// TIA Portal V20 export
// export: Created 2025-12-01T14:57:14.0359159Z, ExportSetting None, DisplayName Totally Integrated Automation Portal, DisplayVersion V20 Update 3, DisplayName TIA Portal Openness, DisplayVersion V20 Update 3, DisplayName TIA Portal Version Control Interface, DisplayVersion V20 Update 3, DisplayName STEP 7 Professional, DisplayVersion V20 Update 3, DisplayName STEP 7 Safety, DisplayVersion V20 Update 2, DisplayName WinCC Basic/Comfort/Advanced, DisplayVersion V20 Update 3, DisplayName WinCC Professional, DisplayVersion V20 Update 3, DisplayName WinCC Unified, DisplayVersion V20 Update 3
FUNCTION "FC810_EventosRecibidos" : Void   // FC810, LAD
TITLE = "Eventos Recibidos" - Tratamiento de los Eventos
{ S7_Optimized_Access := 'FALSE' }
AUTHOR : TRACKING
NAME : 20170707
VERSION : 4.5
// stored: AutoNumber false, SetENOAutomatically false
   VAR_INPUT
      NumJDT : UInt;
   END_VAR
   VAR_TEMP
      AtributosDeUTs : Struct   // Atributos Recibidos de las UTs
         Ruta : Array[0..20] of UInt;   // Ruta Recibida
         Etiqueta : Array[0..42] of Char;   // Etiqueta
         QUBIQA_PID : Array[0..20] of Char;   // QUBIQA - PID del Bulto
         CambiarUTDeMesa : Struct
            Origen : UInt;
            Destino : UInt;
            NOK : Bool;
            OK : Bool;
            Inicio : Bool;
            Final : Bool;
         END_STRUCT;
         AtributosTipoDeCarga : Struct
            Vacia : Bool;
            Pila : Bool;
            Remontada : Bool;
         END_STRUCT;
         Mckey : UDInt;   // Mckey
         MesaActual : UInt;   // Mesa Actual
         MesaDestino : UInt;   // Mesa Destino
         MesaIntermedia : UInt;   // Mesa Intermedia
         OrdenSalida : UInt;   // Orden de Salida
         TipoCarga : USInt;   // **** Tipo de la Carga
         Grupo : UInt;   // Grupo
         CantidadGrupo : USInt;   // Cantidad del Grupo
         PosicionGrupo : USInt;   // Posicion del Grupo
         CodigoFlejado : USInt;   // Codigo de Flejado
         CodigoEnfardado : USInt;   // Codigo de Enfradado
         CodigoEtiquetado : USInt;   // Codigo de Etiquetado
         GaliboAltura : USInt;   // Galibo - Codigo de Altura
         GaliboAnchura : USInt;   // Galibo - Codigo de Anchura
         GaliboProfundidad : USInt;   // Galibo - Codigo de Profundidad
         GaliboTaco : USInt;   // Galibo - Codigo de Taco
         GaliboHueco : USInt;   // Galibo - Codigo de Hueco
         GaliboHuecoRemontada : USInt;   // Galibo - Codigo de Hueco de Carga Remontada
         GaliboColor : USInt;   // Galibo - Codigo de Color de la Carga
         GaliboPatin : USInt;   // Galibo - Codigo de Patin
         GaliboSGA : USInt;   // Galibo - Codigo de SGA
         Presion : UInt;   // Presion de DesPaletizado o Paletizaado de Cajas de Plastico
         CotaAmarre : UInt;   // Cota de Amarre de Cajas de Plastico
         CotaAltura : UInt;   // Cota de la Altura
         CotaAnchura : UInt;   // Cota de la Anchura
         CotaProfundidad : UInt;   // Cota de la Profundidad
         Peso : UDInt;   // Peso
         PosicionDeLaEtiqueta : UInt;   // Posicion Actual de la Etiqueta
         QUBIQA_NumeroBulto : UInt;   // QUBIQA - Numero de Bulto
         QUBIQA_TotalBultos : UInt;   // QUBIQA - Numero Total de Bultos
      END_STRUCT;
      AtributosDeDispositivos : Struct   // Atributos Recibidos del Dispositivo
         TextoRecibido : Array[0..50] of Char;
         MotivoDelError : Array[0..50] of Char;   // TEXTO - Motivo del Error
         BalizaColor : "UDT_DatosBaliza";
         Tipo : UInt;   // Tipo
         Numero : UInt;   // Numero
         NuevoEstado : UInt;   // NuevoEstado
         Habilitado : UInt;
         Prioridad : UInt;
         Operacion : UInt;
         MesaHorquilla : UInt;
         MesaCargaDesCarga : UInt;
      END_STRUCT;
      VarTempUTs : Struct
         Mckey : UDInt;
         MesaActual : UInt;
         NumeroUT : UInt;
         SalidaEventoRETI : UInt;
      END_STRUCT;
      VarTempDispositivos : Struct
         Baliza : "UDT_DatosBaliza";
         Numero : UInt;
      END_STRUCT;
      DBEventosRec : Word;   // DB de Eventos Recibidos
      P_Eventos : DWord;   // Puntero al DB de Eventos Recibidos
      Evento : DWord;   // Etiqueta - Evento
      Atributo : DWord;   // Etiqueta - Atributo
      EtiquetaAtributo : DWord;   // Etiqueta - Conversion de Atributo
      NumeroEvento : UInt;   // Numero de Evento
      NumeroAtributo : UInt;   // Numero de Atributo
      Leido : UInt;
      ValorDeAtributo : UDInt;   // Valor del Atributo
      ValorDeEtiqueta : UInt;   // Valor de la Etiqueta - Conversion de Atributo
      Indice : UInt;   // Indice en el recorrido de los ARRAYs
      IndiceCBOX : UInt;
      IndiceVTDC : UInt;
      IndiceMesa : UInt;
      IndiceMaquina : UInt;
      IndiceDispositivosVarios : UInt;
      OffsetInicial : UInt;
      LonguitudTextoRecibido : UInt;
      ReturnValor : Int;
      Cero : Byte;
      JDT02_Activo : Bool;
      MesaDeJDT02 : Bool;
      DispositivoDeJDT02 : Bool;
   END_VAR
BEGIN

NETWORK
TITLE = Inicializar
/////////////////////////////////////////////////////////////////////////
/// --- Comprobar que JDT

      SET;
      R     #JDT02_Activo;
      L     "JDT1_NDB_EventosRec";  // Cogemos el DB de Eventos Recibidos
      T     #DBEventosRec;

/////////////////////////////////////////////////////////////////////////

      L     #NumJDT;
      L     2;
      <>I;
      JC    NoJdT02;

/////////////////////////////////////////////////////////////////////////

      SET;
      S     #JDT02_Activo;
      L     "JDT2_NDB_EventosRec";  // Cogemos el DB de Eventos Recibidos
      T     #DBEventosRec;

NoJdT02:NOP   0;

/////////////////////////////////////////////////////////////////////////



NETWORK
TITLE = Analizar la lista de Eventos
/////////////////////////////////////////////////////////////////////////
// Inicializar el Puntero de la Lista de Eventos

      L     0;  // Inicializar el Puntero de Eventos
      LAR2;

      OPN   DB [#DBEventosRec];  // Mirar si tiene algo el DB de Eventos Recibidos
      L     DBB [AR2, P#0.0];
      L     0;
      ==I;
      JC    NoLimpiarNada;


/////////////////////////////////////////////////////////////////////////
InicioBucle_EventosRecibidos:NOP   0;
      OPN   DB [#DBEventosRec];  // Leer el digito de Eventos Recibidos
      L     DBB [AR2, P#0.0];
      T     #Leido;

// Buscando Principio de Evento

      L     #Leido;
      L     '{';  // Inicio de Evento - '{'
      ==I;
      JC    EventosRecibidos;  // Tratar el Nuevo Evento

// Buscando el Final de la Lista de Eventos

      L     #Leido;
      L     3;  // Final de la Lista de Eventos - 0x03
      ==I;
      JC    FinalizarFuncion;  // Finalizar, ya no hay más Eventos
      L     #Leido;
      L     0;  // Final de la Lista de Eventos - 0x00 - No hay Mas
      ==I;
      JC    FinalizarFuncion;  // Finalizar, ya no hay más Eventos


/////////////////////////////////////////////////////////////////////////
FinBucle_EventosRecibidos:NOP   0;
      +AR2  P#1.0;  // Seguir recorriendo la Lista de Eventos
      JU    InicioBucle_EventosRecibidos;



NETWORK
TITLE = Distribucion de los Eventos (LIsta del DB de Conversion)
EventosRecibidos:NOP   0;

/////////////////////////////////////////////////////////////////////////
/////////////////////////////////////////////////////////////////////////
/////////////////////////////////////////////////////////////////////////
// Hay que recoger el Evento, para despues repartir
// Despues '{' va el tipo de eventos (2 Bytes)

      +AR2  P#1.0;
      OPN   DB [#DBEventosRec];
      L     DBD [AR2, P#0.0];  // Recogo el tipo de Evento (4 Caracteres)
      T     #Evento;


/////////////////////////////////////////////////////////////////////////
/////////////////////////////////////////////////////////////////////////
/////////////////////////////////////////////////////////////////////////
// Buscar numero de evento
      L     1;
      T     #NumeroEvento;
BucleDeBusqueda_NumeroDeEvento:NOP   0;

// -- Se ha encontrado el Evento Recibido
      L     "DB870_ConversorEventos".EventosRecibidos[#NumeroEvento];
      L     #Evento;
      ==D;
      JC    Encontrado_NumeroDeEvento;

// -- Final de la lista de Eventos Recibidos - No Encontrado
      L     "DB870_ConversorEventos".EventosRecibidos[#NumeroEvento];
      L     0;
      ==D;
      JC    InicioBucle_EventosRecibidos;

// --- Maximo del Array de la Lista de Eventos Recibidos - No Encontrado
      L     #NumeroEvento;
      L     "CTE_MaxArrayConversion";
      >=I;
      JC    InicioBucle_EventosRecibidos;

// --- Continuar la Busqueda
      L     #NumeroEvento;
      L     1;
      +I;
      T     #NumeroEvento;
      JU    BucleDeBusqueda_NumeroDeEvento;



NETWORK
TITLE = ----
/////////////////////////////////////////////////////////////////////////
/////////////////////////////////////////////////////////////////////////
/////////////////////////////////////////////////////////////////////////
// Distribuir dependiendo del Resultado de la Busqueda del Evento Recibido
// Para recoger los Atributos
Encontrado_NumeroDeEvento:NOP   0;
      L     #NumeroEvento;
      JL    NoExiste_NumeroDeEvento;

      JU    NoExiste_NumeroDeEvento;
      JU    Atributos_EventosDeLasUTs;  // Evento (01) - CREA
      JU    Atributos_EventosDeLasUTs;  // Evento (02) - RUTA
      JU    Atributos_EventosDeLasUTs;  // Evento (03) - DRUT
      JU    Atributos_EventosDeLasUTs;  // Evento (04) - RETI
      JU    Atributos_EventosDeLasUTs;  // Evento (05) - BORR
      JU    Atributos_EventosDeLasUTs;  // Evento (06) - DATA
      JU    Atributos_EventosDeLasUTs;  // Evento (07) - ?UT?
      JU    Atributos_EventosDeLasUTs;  // Evento (08) - MOVE
      JU    Atributos_EventosDeLasUTs;  // Evento (09) - DEMB

      JU    Atributos_EventosDeLosDispositivos;  // Evento (10) - CSTA
      JU    Atributos_EventosDeLosDispositivos;  // Evento (11) - DIDO

      JU    EventosRecibidos_Router;  // Evento (12) - ORDE
      JU    EventosRecibidos_Router;  // Evento (13) - BOET
      JU    EventosRecibidos_Router;  // Evento (14) - BOBD
      JU    EventosRecibidos_Router;  // Evento (15) - RUET
      JU    EventosRecibidos_Router;  // Evento (16) - RUES
      JU    EventosRecibidos_Router;  // Evento (17) - INIR

      JU    Atributos_EventosDeLosDispositivos;  // Evento (18) - ?ST?

      JU    EventosRecibidos_Quimarox;  // Evento (19) - QCRE
      JU    EventosRecibidos_Quimarox;  // Evento (20) - QPR?

      JU    EventosRecibidos_Reset_V2;  // Evento (21) - CHEQ

/////////////////////////////////////////////////////////////////////////
NoExiste_NumeroDeEvento:NOP   0;
      JU    InicioBucle_EventosRecibidos;



NETWORK
TITLE = Analizar la lista de los Atributos de las UTs
Atributos_EventosDeLasUTs:NOP   0;

/////////////////////////////////////////////////////////////////////////
/////////////////////////////////////////////////////////////////////////
/////////////////////////////////////////////////////////////////////////
// Inicializa variables de los Atributos de las UTs
      L     0;
      T     #Cero;

      CALL  FILL
      ( BVAL    := #Cero,
        RET_VAL := #ReturnValor,
        BLK     := #AtributosDeUTs
      );  // Inicializa Atributos de las UTS



NETWORK
TITLE = ----
/////////////////////////////////////////////////////////////////////////
/////////////////////////////////////////////////////////////////////////
// Buscando Atributos o Final del Evento
      +AR2  P#4.0;  // Prepara Puntero para ver los atributos

InicioBucleAtributos_EventosDeLasUTs:NOP   0;
      OPN   DB [#DBEventosRec];
      L     DBB [AR2, P#0.0];
      T     #Leido;

// Inicio de atributo - Ir a tratar los atributos
      L     #Leido;
      L     '[';  // '[' - Inicio de Atributo
      ==I;  // Atributo del Evento
      JC    EncontradoAtributos_EventosDeLasUTs;

// Fin del Evento
      L     #Leido;
      L     '}';  // '}' - Fin del Evento
      ==I;  // Se acabo el evento
      JC    FinalAtributos_EventosDeLasUTs;

// Sin Mensaje
      L     #Leido;
      L     0;  // No hay mas Mensaje
      ==I;  // Se acabo el evento
      JC    FinalAtributos_EventosDeLasUTs;


      +AR2  P#1.0;  // Seguir buscado atributo
      JU    InicioBucleAtributos_EventosDeLasUTs;


/////////////////////////////////////////////////////////////////////////
/////////////////////////////////////////////////////////////////////////
// Se acaba el Evento - Ir a guardar datos del Evento
FinalAtributos_EventosDeLasUTs:NOP   0;
      TAR2;
      T     #P_Eventos;  // Guardo Por donde voy en la lista de eventos
      JU    GuardarDatos_EventosRecibidos;



NETWORK
TITLE = Distribucion de los Atributos de las UTs (LIsta del DB de Conversion)
EncontradoAtributos_EventosDeLasUTs:NOP   0;

/////////////////////////////////////////////////////////////////////////
/////////////////////////////////////////////////////////////////////////
/////////////////////////////////////////////////////////////////////////
/////////////////////////////////////////////////////////////////////////
// Mirar que Atributo del Evento  es ?
      +AR2  P#1.0;
      OPN   DB [#DBEventosRec];
      L     DBD [AR2, P#0.0];  // Atributo - 4 Caracteres
      T     #Atributo;

/////////////////////////////////////////////////////////////////////////
/////////////////////////////////////////////////////////////////////////
/////////////////////////////////////////////////////////////////////////
// Buscar numero de Atributo
      L     1;
      T     #NumeroAtributo;
BucleDeBusqueda_NumeroDeAtributoDeUTs:NOP   0;

// -- Se ha encontrado el Atributo Recibido
      L     "DB870_ConversorEventos".AtributosRecibidosDeUTs[#NumeroAtributo];
      L     #Atributo;
      ==D;
      JC    Encontrado_NumeroDeAtributoDeUTs;

// -- Final de la lista de Atributo Recibidos - No Encontrado
      L     "DB870_ConversorEventos".AtributosRecibidosDeUTs[#NumeroAtributo];
      L     0;
      ==D;
      JC    InicioBucleAtributos_EventosDeLasUTs;

// --- Maximo del Array de la Lista de Atributo Recibidos - No Encontrado
      L     #NumeroAtributo;
      L     "CTE_MaxArrayConversion";
      >=I;
      JC    InicioBucleAtributos_EventosDeLasUTs;


// --- Continuar la Busqueda
      L     #NumeroAtributo;
      L     1;
      +I;
      T     #NumeroAtributo;
      JU    BucleDeBusqueda_NumeroDeAtributoDeUTs;



NETWORK
TITLE = ----
/////////////////////////////////////////////////////////////////////////
/////////////////////////////////////////////////////////////////////////
/////////////////////////////////////////////////////////////////////////
// Distribuir dependiendo del Resultado de la Busqueda de Atributo Recibido
Encontrado_NumeroDeAtributoDeUTs:NOP   0;
      L     #NumeroAtributo;
      JL    NoExiste_NumeroDeAtibutoDeUTs;

      JU    NoExiste_NumeroDeAtibutoDeUTs;
      JU    AtributoDeUTs_MCKY;  // Atributo (01) - MCKY
      JU    AtributoDeUTs_MESA;  // Atributo (02) - MESA
      JU    AtributoDeUTs_RUTA;  // Atributo (03) - RUTA
      JU    AtributoDeUTs_SALI;  // Atributo (04) - SALI
      JU    AtributoDeUTs_SSCC;  // Atributo (05) - SSCC

      JU    AtributoDeUTs_GRUP;  // Atributo (06) - GRUP
      JU    AtributoDeUTs_GCNT;  // Atributo (07) - GCNT
      JU    AtributoDeUTs_GORD;  // Atributo (08) - GORD

      JU    AtributoDeUTs_FLEJ;  // Atributo (09) - FLEJ
      JU    AtributoDeUTs_ENFA;  // Atributo (10) - ENFA
      JU    AtributoDeUTs_ETIQ;  // Atributo (11) - ETIQ

      JU    AtributoDeUTs_AMAR;  // Atributo (12) - AMAR
      JU    AtributoDeUTs_PRES;  // Atributo (13) - PRES

      JU    AtributoDeUTs_NBUL_QUBIQA;  // Atributo (14) - NBUL (QUBIQA)
      JU    AtributoDeUTs_NTBU_QUBIQA;  // Atributo (15) - NTBU (QUBIQA)
      JU    AtributoDeUTs_PID_QUBIQA;  // Atributo (16) - PID_ (QUBIQA)

      JU    AtributoDeUTs_TIPO;  // Atributo (17) - TIPO
      JU    AtributoDeUTs_REMO;  // Atributo (18) - REMO
      JU    AtributoDeUTs_PILA;  // Atributo (19) - PILA
      JU    AtributoDeUTs_VACI;  // Atributo (20) - VACI

      JU    AtributoDeUTs_COTA;  // Atributo (21) - COTA
      JU    AtributoDeUTs_COTW;  // Atributo (22) - COTW
      JU    AtributoDeUTs_COTL;  // Atributo (23) - COTL
      JU    AtributoDeUTs_PESO;  // Atributo (24) - PESO

      JU    AtributoDeUTs_ALTO;  // Atributo (25) - ALTO
      JU    AtributoDeUTs_ANCH;  // Atributo (26) - ANCH
      JU    AtributoDeUTs_PROF;  // Atributo (27) - PROF
      JU    AtributoDeUTs_TACO;  // Atributo (28) - TACO
      JU    AtributoDeUTs_HUEC;  // Atributo (29) - HUEC
      JU    AtributoDeUTs_HUER;  // Atributo (30) - HUER
      JU    AtributoDeUTs_COLO;  // Atributo (31) - COLO
      JU    AtributoDeUTs_PATI;  // Atributo (32) - PATI

      JU    AtributoDeUTs_LETI;  // Atributo (33) - LETI

      JU    AtributoDeUTs_SGAP;  // Atributo (34) - SGAP
      JU    AtributoDeUTs_SGAE;  // Atributo (35) - SGAE
      JU    AtributoDeUTs_SGAD;  // Atributo (36) - SGAD
      JU    AtributoDeUTs_SGA_Error;  // Atributo (37) - SGA

      JU    AtributoDeUTs_RSLT;  // Atributo (38) - RSLT
      JU    AtributoDeUTs_PDST;  // Atributo (39) - PDST
      JU    AtributoDeUTs_DEST;  // Atributo (40) - DEST

      JU    AtributoDeUTs_FLEJ;  // Atributo (41) - PALE >>> NDD

/////////////////////////////////////////////////////////////////////////
NoExiste_NumeroDeAtibutoDeUTs:NOP   0;
      JU    InicioBucleAtributos_EventosDeLasUTs;



NETWORK
TITLE = ---- ---- Recoger el Atributo de las UTs - MCKY
/////////////////////////////////////////////////////////////////////////
/////////////////////////////////////////////////////////////////////////
/////////////////////////////////////////////////////////////////////////
AtributoDeUTs_MCKY:NOP   0;
      +AR2  P#5.0;
      TAR2;
      T     #P_Eventos;
      SRD   3;
      T     #OffsetInicial;

// Obtener el Valor del Atributo
      CALL  "FC892_Obtener_ValorDelAtributo"
      ( DB_String := #DBEventosRec,
        OffsetIni := #OffsetInicial,
        Valor     := #ValorDeAtributo
      );

      L     #ValorDeAtributo;  // Lo guardo
      T     #AtributosDeUTs.Mckey;

// Continuo con el Evento
      L     #P_Eventos;
      LAR2;
      JU    InicioBucleAtributos_EventosDeLasUTs;



NETWORK
TITLE = ---- ---- Recoger el Atributo de las UTs - MESA
/////////////////////////////////////////////////////////////////////////
/////////////////////////////////////////////////////////////////////////
/////////////////////////////////////////////////////////////////////////
AtributoDeUTs_MESA:NOP   0;
      +AR2  P#5.0;
      TAR2;
      T     #P_Eventos;
      SRD   3;
      T     #OffsetInicial;

// Obtener el Valor del Atributo
      CALL  "FC892_Obtener_ValorDelAtributo"
      ( DB_String := #DBEventosRec,
        OffsetIni := #OffsetInicial,
        Valor     := #ValorDeAtributo
      );

      L     #ValorDeAtributo;  // Lo guardo
      T     #AtributosDeUTs.MesaActual;

// Continuo con el Evento
      L     #P_Eventos;
      LAR2;
      JU    InicioBucleAtributos_EventosDeLasUTs;



NETWORK
TITLE = ---- ---- Recoger el Atributo de las UTs - RUTA
/////////////////////////////////////////////////////////////////////////
/////////////////////////////////////////////////////////////////////////
/////////////////////////////////////////////////////////////////////////
AtributoDeUTs_RUTA:NOP   0;
      +AR2  P#5.0;  // Preparo punteros
      L     0;
      T     #Indice;

/////////////////////////////////////////////////////////////////////////
// Inicio para recoger la nueva ruta
InicioBucleAtributoDeUTs_RUTA:NOP   0;
      OPN   DB [#DBEventosRec];
      L     DBB [AR2, P#0.0];
      T     #Leido;

// Mirar si es nueva mesa o final de ruta

      L     #Leido;
      L     '[';  // Nueva ruta de la Mesa
      ==I;
      JC    NuevaMesaAtributoDeUTs_RUTA;
      L     #Leido;
      L     ')';  // Es Final de Ruta
      ==I;
      JC    FinalBucleAtributoDeUTs_RUTA;

      +AR2  P#1.0;  // Continuar hasta encontrar otra Mesa de la ruta
      JU    InicioBucleAtributoDeUTs_RUTA;


/////////////////////////////////////////////////////////////////////////
// Nueva mesa para la ruta, recogerla y guradarla
NuevaMesaAtributoDeUTs_RUTA:NOP   0;
      +AR2  P#6.0;
      TAR2;
      T     #P_Eventos;
      SRD   3;
      T     #OffsetInicial;

// Obtener el Valor de la Mesa de la Ruta

      CALL  "FC892_Obtener_ValorDelAtributo"
      ( DB_String := #DBEventosRec,
        OffsetIni := #OffsetInicial,
        Valor     := #ValorDeAtributo
      );
      L     #ValorDeAtributo;  // Lo guardo
      T     #AtributosDeUTs.Ruta[#Indice];
      T     #AtributosDeUTs.MesaDestino;

      L     #Indice;  // Siguiente Mesa de la Ruta
      L     1;
      +I;
      T     #Indice;

      L     0;  //Se pone a 0 para indicar final de ruta
      T     #AtributosDeUTs.Ruta[#Indice];

      L     #P_Eventos;
      LAR2;
      JU    InicioBucleAtributoDeUTs_RUTA;


/////////////////////////////////////////////////////////////////////////
// No tiene más mesas la ruta. Continuo con el Evento
FinalBucleAtributoDeUTs_RUTA:NOP   0;
      L     #AtributosDeUTs.Ruta[0];  // Mesa Intermedia la primera mesa de la Ruta
      T     #AtributosDeUTs.MesaIntermedia;

      L     #P_Eventos;
      LAR2;
      JU    InicioBucleAtributos_EventosDeLasUTs;



NETWORK
TITLE = ---- ---- Recoger el Atributo de las UTs - SALI
/////////////////////////////////////////////////////////////////////////
/////////////////////////////////////////////////////////////////////////
/////////////////////////////////////////////////////////////////////////
AtributoDeUTs_SALI:NOP   0;
      +AR2  P#5.0;
      TAR2;
      T     #P_Eventos;
      SRD   3;
      T     #OffsetInicial;

// Obtener el Valor del Atributo
      CALL  "FC892_Obtener_ValorDelAtributo"
      ( DB_String := #DBEventosRec,
        OffsetIni := #OffsetInicial,
        Valor     := #ValorDeAtributo
      );

      L     #ValorDeAtributo;  // Lo guardo
      T     #AtributosDeUTs.OrdenSalida;

// Continuo con el Evento
      L     #P_Eventos;
      LAR2;
      JU    InicioBucleAtributos_EventosDeLasUTs;



NETWORK
TITLE = ---- ---- Recoger el Atributo de las UTs - SSCC
/////////////////////////////////////////////////////////////////////////
/////////////////////////////////////////////////////////////////////////
/////////////////////////////////////////////////////////////////////////
AtributoDeUTs_SSCC:NOP   0;
      +AR2  P#5.0;
      L     2;
      T     #Indice;

/////////////////////////////////////////////////////////////////////////
// Inicio a recoger la etiqueta
InicioBucleAtributoDeUTs_Etiqueta:NOP   0;
      OPN   DB [#DBEventosRec];
      L     DBB [AR2, P#0.0];
      T     #Leido;

      L     #Leido;
      L     '}';  // Es Final de etiqueta
      ==I;
      JC    FinalBucleAtributoDeUTs_Etiqueta;
      L     #Leido;
      L     '[';  // Es Final de etiqueta
      ==I;
      JC    FinalBucleAtributoDeUTs_Etiqueta;

      L     #Leido;
      T     #AtributosDeUTs.Etiqueta[#Indice];

      L     #Indice;  // Siguiente caracter
      L     1;
      +I;
      T     #Indice;
      +AR2  P#1.0;

      L     0;
      T     #AtributosDeUTs.Etiqueta[#Indice];
      JU    InicioBucleAtributoDeUTs_Etiqueta;

/////////////////////////////////////////////////////////////////////////
FinalBucleAtributoDeUTs_Etiqueta:NOP   0;
      L     40;  // Inicio la carcacteristica de la STRING
      T     #AtributosDeUTs.Etiqueta[0];
      L     #Indice;
      L     2;
      -I;
      T     #AtributosDeUTs.Etiqueta[1];

      JU    InicioBucleAtributos_EventosDeLasUTs;



NETWORK
TITLE = ---- ---- Recoger el Atributo de las UTs - GRUP
/////////////////////////////////////////////////////////////////////////
/////////////////////////////////////////////////////////////////////////
/////////////////////////////////////////////////////////////////////////
AtributoDeUTs_GRUP:NOP   0;
      +AR2  P#5.0;
      TAR2;
      T     #P_Eventos;
      SRD   3;
      T     #OffsetInicial;

// Obtener el Valor del Atributo
      CALL  "FC892_Obtener_ValorDelAtributo"
      ( DB_String := #DBEventosRec,
        OffsetIni := #OffsetInicial,
        Valor     := #ValorDeAtributo
      );

      L     #ValorDeAtributo;  // Lo guardo
      T     #AtributosDeUTs.Grupo;

// Continuo con el Evento
      L     #P_Eventos;
      LAR2;
      JU    InicioBucleAtributos_EventosDeLasUTs;



NETWORK
TITLE = ---- ---- Recoger el Atributo de las UTs - GCNT (Cantidad de UTs en el Grupo)
/////////////////////////////////////////////////////////////////////////
/////////////////////////////////////////////////////////////////////////
/////////////////////////////////////////////////////////////////////////
AtributoDeUTs_GCNT:NOP   0;
      +AR2  P#5.0;
      TAR2;
      T     #P_Eventos;
      SRD   3;
      T     #OffsetInicial;

// Obtener el Valor del Atributo
      CALL  "FC892_Obtener_ValorDelAtributo"
      ( DB_String := #DBEventosRec,
        OffsetIni := #OffsetInicial,
        Valor     := #ValorDeAtributo
      );

      L     #ValorDeAtributo;  // Lo guardo
      T     #AtributosDeUTs.CantidadGrupo;

// Continuo con el Evento
      L     #P_Eventos;
      LAR2;
      JU    InicioBucleAtributos_EventosDeLasUTs;



NETWORK
TITLE = ---- ---- Recoger el Atributo de las UTs - GORD (Posicion en el Grupo)
/////////////////////////////////////////////////////////////////////////
/////////////////////////////////////////////////////////////////////////
/////////////////////////////////////////////////////////////////////////
AtributoDeUTs_GORD:NOP   0;
      +AR2  P#5.0;
      TAR2;
      T     #P_Eventos;
      SRD   3;
      T     #OffsetInicial;

// Obtener el Valor del Atributo
      CALL  "FC892_Obtener_ValorDelAtributo"
      ( DB_String := #DBEventosRec,
        OffsetIni := #OffsetInicial,
        Valor     := #ValorDeAtributo
      );

      L     #ValorDeAtributo;  // Lo guardo
      T     #AtributosDeUTs.PosicionGrupo;

// Continuo con el Evento
      L     #P_Eventos;
      LAR2;
      JU    InicioBucleAtributos_EventosDeLasUTs;



NETWORK
TITLE = ---- ---- Recoger el Atributo de las UTs - FLEJ (Codigo de Flejado)
/////////////////////////////////////////////////////////////////////////
/////////////////////////////////////////////////////////////////////////
/////////////////////////////////////////////////////////////////////////
AtributoDeUTs_FLEJ:NOP   0;
      +AR2  P#5.0;
      TAR2;
      T     #P_Eventos;
      SRD   3;
      T     #OffsetInicial;

// Obtener el Valor del Atributo
      CALL  "FC892_Obtener_ValorDelAtributo"
      ( DB_String := #DBEventosRec,
        OffsetIni := #OffsetInicial,
        Valor     := #ValorDeAtributo
      );

      L     #ValorDeAtributo;  // Lo guardo
      T     #AtributosDeUTs.CodigoFlejado;

// Continuo con el Evento
      L     #P_Eventos;
      LAR2;
      JU    InicioBucleAtributos_EventosDeLasUTs;



NETWORK
TITLE = ---- ---- Recoger el Atributo de las UTs - ENFA (Codigo de Enfardado)
/////////////////////////////////////////////////////////////////////////
/////////////////////////////////////////////////////////////////////////
/////////////////////////////////////////////////////////////////////////
AtributoDeUTs_ENFA:NOP   0;
      +AR2  P#5.0;
      TAR2;
      T     #P_Eventos;
      SRD   3;
      T     #OffsetInicial;

// Obtener el Valor del Atributo
      CALL  "FC892_Obtener_ValorDelAtributo"
      ( DB_String := #DBEventosRec,
        OffsetIni := #OffsetInicial,
        Valor     := #ValorDeAtributo
      );

      L     #ValorDeAtributo;  // Lo guardo
      T     #AtributosDeUTs.CodigoEnfardado;

// Continuo con el Evento
      L     #P_Eventos;
      LAR2;
      JU    InicioBucleAtributos_EventosDeLasUTs;



NETWORK
TITLE = ---- ---- Recoger el Atributo de las UTs - ETIQ (Codigo de Etiquetado)
/////////////////////////////////////////////////////////////////////////
/////////////////////////////////////////////////////////////////////////
/////////////////////////////////////////////////////////////////////////
AtributoDeUTs_ETIQ:NOP   0;
      +AR2  P#5.0;
      TAR2;
      T     #P_Eventos;
      SRD   3;
      T     #OffsetInicial;

// Obtener el Valor del Atributo
      CALL  "FC892_Obtener_ValorDelAtributo"
      ( DB_String := #DBEventosRec,
        OffsetIni := #OffsetInicial,
        Valor     := #ValorDeAtributo
      );

      L     #ValorDeAtributo;  // Lo guardo
      T     #AtributosDeUTs.CodigoEtiquetado;

// Continuo con el Evento
      L     #P_Eventos;
      LAR2;
      JU    InicioBucleAtributos_EventosDeLasUTs;



NETWORK
TITLE = ---- ---- Recoger el Atributo de las UTs - AMAR (Cota de Amarre de las Cajas de Plastico)
/////////////////////////////////////////////////////////////////////////
/////////////////////////////////////////////////////////////////////////
/////////////////////////////////////////////////////////////////////////
AtributoDeUTs_AMAR:NOP   0;
      +AR2  P#5.0;
      TAR2;
      T     #P_Eventos;
      SRD   3;
      T     #OffsetInicial;

// Obtener el Valor del Atributo
      CALL  "FC892_Obtener_ValorDelAtributo"
      ( DB_String := #DBEventosRec,
        OffsetIni := #OffsetInicial,
        Valor     := #ValorDeAtributo
      );

      L     #ValorDeAtributo;  // Lo guardo
      T     #AtributosDeUTs.CotaAmarre;

// Continuo con el Evento
      L     #P_Eventos;
      LAR2;
      JU    InicioBucleAtributos_EventosDeLasUTs;



NETWORK
TITLE = ---- ---- Recoger el Atributo de las UTs - PRES (Presion para el Paletizador y DesPaletizador de las Cajas de Plastico) /// OJOOOOOOO
/////////////////////////////////////////////////////////////////////////
/////////////////////////////////////////////////////////////////////////
/////////////////////////////////////////////////////////////////////////
AtributoDeUTs_PRES:NOP   0;
      +AR2  P#5.0;
      TAR2;
      T     #P_Eventos;
      SRD   3;
      T     #OffsetInicial;

// Obtener el Valor del Atributo
      CALL  "FC892_Obtener_ValorDelAtributo"
      ( DB_String := #DBEventosRec,
        OffsetIni := #OffsetInicial,
        Valor     := #ValorDeAtributo
      );

      L     #ValorDeAtributo;  // Lo guardo
      T     #AtributosDeUTs.Presion;

// Continuo con el Evento
      L     #P_Eventos;
      LAR2;
      JU    InicioBucleAtributos_EventosDeLasUTs;



NETWORK
TITLE = ---- ---- Recoger el Atributo de las UTs - NBUL (QUBIQA - Nurmero de Bulto)
/////////////////////////////////////////////////////////////////////////
/////////////////////////////////////////////////////////////////////////
/////////////////////////////////////////////////////////////////////////
AtributoDeUTs_NBUL_QUBIQA:NOP   0;
      +AR2  P#5.0;
      TAR2;
      T     #P_Eventos;
      SRD   3;
      T     #OffsetInicial;

// Obtener el Valor del Atributo
      CALL  "FC892_Obtener_ValorDelAtributo"
      ( DB_String := #DBEventosRec,
        OffsetIni := #OffsetInicial,
        Valor     := #ValorDeAtributo
      );

      L     #ValorDeAtributo;  // Lo guardo
      T     #AtributosDeUTs.QUBIQA_NumeroBulto;

// Continuo con el Evento
      L     #P_Eventos;
      LAR2;
      JU    InicioBucleAtributos_EventosDeLasUTs;



NETWORK
TITLE = ---- ---- Recoger el Atributo de las UTs - NTBU (QUBIQA - Numerom Total de Bultos)
/////////////////////////////////////////////////////////////////////////
/////////////////////////////////////////////////////////////////////////
/////////////////////////////////////////////////////////////////////////
AtributoDeUTs_NTBU_QUBIQA:NOP   0;
      +AR2  P#5.0;
      TAR2;
      T     #P_Eventos;
      SRD   3;
      T     #OffsetInicial;

// Obtener el Valor del Atributo
      CALL  "FC892_Obtener_ValorDelAtributo"
      ( DB_String := #DBEventosRec,
        OffsetIni := #OffsetInicial,
        Valor     := #ValorDeAtributo
      );

      L     #ValorDeAtributo;  // Lo guardo
      T     #AtributosDeUTs.QUBIQA_TotalBultos;

// Continuo con el Evento
      L     #P_Eventos;
      LAR2;
      JU    InicioBucleAtributos_EventosDeLasUTs;



NETWORK
TITLE = ---- ---- Recoger el Atributo de las UTs - PID_ (QIBIQA - PID del Bulto - 20 Caracteres)
/////////////////////////////////////////////////////////////////////////
/////////////////////////////////////////////////////////////////////////
/////////////////////////////////////////////////////////////////////////
AtributoDeUTs_PID_QUBIQA:NOP   0;
      +AR2  P#5.0;
      L     0;
      T     #Indice;

/////////////////////////////////////////////////////////////////////////
// Inicio a recoger la etiqueta
InicioBucleAtributoDeUTs_PID_QUBIQA:NOP   0;
      OPN   DB [#DBEventosRec];
      L     DBB [AR2, P#0.0];
      T     #Leido;

      L     #Leido;
      L     '}';  // Es Final de etiqueta
      ==I;
      JC    FinalBucleAtributoDeUTs_PID_QUBIQA;
      L     #Leido;
      L     '[';  // Es Final de etiqueta
      ==I;
      JC    FinalBucleAtributoDeUTs_PID_QUBIQA;

      L     #Leido;
      T     #AtributosDeUTs.QUBIQA_PID[#Indice];

      L     #Indice;  // Siguiente caracter
      L     1;
      +I;
      T     #Indice;
      +AR2  P#1.0;

      L     0;
      T     #AtributosDeUTs.QUBIQA_PID[#Indice];
      JU    InicioBucleAtributoDeUTs_PID_QUBIQA;

/////////////////////////////////////////////////////////////////////////
FinalBucleAtributoDeUTs_PID_QUBIQA:NOP   0;
      JU    InicioBucleAtributos_EventosDeLasUTs;



NETWORK
TITLE = ---- ---- Recoger el Atributo de las UTs - TIPO (Tipo de Carga) ****
/////////////////////////////////////////////////////////////////////////
/////////////////////////////////////////////////////////////////////////
/////////////////////////////////////////////////////////////////////////
AtributoDeUTs_TIPO:NOP   0;
      +AR2  P#5.0;

      OPN   DB [#DBEventosRec];
      L     DBD [AR2, P#0.0];
      T     #EtiquetaAtributo;

// Obtener el Valor del Atributo
      CALL  "FC894_Obtener_ValorDeEtiqueta"
      ( EtiquetaEvento := #EtiquetaAtributo,
        ValorEvento    := #ValorDeEtiqueta
      );

      L     #ValorDeEtiqueta;  // Lo guardo
      T     #AtributosDeUTs.TipoCarga;


// Continuo con el Evento
      +AR2  P#4.0;
      JU    InicioBucleAtributos_EventosDeLasUTs;



NETWORK
TITLE = ---- ---- Recoger el Atributo de las UTs - REMO (La Carga esta Remontada)
/////////////////////////////////////////////////////////////////////////
/////////////////////////////////////////////////////////////////////////
/////////////////////////////////////////////////////////////////////////
AtributoDeUTs_REMO:NOP   0;
      +AR2  P#5.0;

      OPN   DB [#DBEventosRec];
      L     DBB [AR2, P#0.0];  // Sacar el Valor del Campo
      T     #Leido;
      +AR2  P#1.0;

      L     #Leido;  // Comparar si es cero
      L     '0';  // La carga No Esta Remontada ?
      ==I;
      JC    InicioBucleAtributos_EventosDeLasUTs;

      SET;
      S     #AtributosDeUTs.AtributosTipoDeCarga.Remontada;


// Continuo con el Evento
      JU    InicioBucleAtributos_EventosDeLasUTs;



NETWORK
TITLE = ---- ---- Recoger el Atributo de las UTs - PILA (La Carga es una Pila)
/////////////////////////////////////////////////////////////////////////
/////////////////////////////////////////////////////////////////////////
/////////////////////////////////////////////////////////////////////////
AtributoDeUTs_PILA:NOP   0;
      +AR2  P#5.0;

      OPN   DB [#DBEventosRec];
      L     DBB [AR2, P#0.0];  // Sacar el Valor del Campo
      T     #Leido;
      +AR2  P#1.0;

      L     #Leido;  // Comparar si es cero
      L     '0';  // La Carga No es Pila
      ==I;
      JC    InicioBucleAtributos_EventosDeLasUTs;

      SET;
      S     #AtributosDeUTs.AtributosTipoDeCarga.Pila;


// Continuo con el Evento
      JU    InicioBucleAtributos_EventosDeLasUTs;



NETWORK
TITLE = ---- ---- Recoger el Atributo de las UTs - VACI ( La carga esta vacia de contenido)
/////////////////////////////////////////////////////////////////////////
/////////////////////////////////////////////////////////////////////////
/////////////////////////////////////////////////////////////////////////
AtributoDeUTs_VACI:NOP   0;
      +AR2  P#5.0;

      OPN   DB [#DBEventosRec];
      L     DBB [AR2, P#0.0];  // Sacar el Valor del Campo
      T     #Leido;
      +AR2  P#1.0;

      L     #Leido;  // Comparar si es cero
      L     '0';  // La carga No esta Vacia
      ==I;
      JC    InicioBucleAtributos_EventosDeLasUTs;

      SET;
      S     #AtributosDeUTs.AtributosTipoDeCarga.Vacia;


// Continuo con el Evento
      JU    InicioBucleAtributos_EventosDeLasUTs;



NETWORK
TITLE = ---- ---- Recoger el Atributo de las UTs - COTA ( Cota de Altura)
/////////////////////////////////////////////////////////////////////////
/////////////////////////////////////////////////////////////////////////
/////////////////////////////////////////////////////////////////////////
AtributoDeUTs_COTA:NOP   0;
      +AR2  P#5.0;
      TAR2;
      T     #P_Eventos;
      SRD   3;
      T     #OffsetInicial;

// Obtener el Valor del Atributo
      CALL  "FC892_Obtener_ValorDelAtributo"
      ( DB_String := #DBEventosRec,
        OffsetIni := #OffsetInicial,
        Valor     := #ValorDeAtributo
      );

      L     #ValorDeAtributo;  // Lo guardo
      T     #AtributosDeUTs.CotaAltura;

// Continuo con el Evento
      L     #P_Eventos;
      LAR2;
      JU    InicioBucleAtributos_EventosDeLasUTs;



NETWORK
TITLE = ---- ---- Recoger el Atributo de las UTs - COTW (Cota de Anchura)
/////////////////////////////////////////////////////////////////////////
/////////////////////////////////////////////////////////////////////////
/////////////////////////////////////////////////////////////////////////
AtributoDeUTs_COTW:NOP   0;
      +AR2  P#5.0;
      TAR2;
      T     #P_Eventos;
      SRD   3;
      T     #OffsetInicial;

// Obtener el Valor del Atributo
      CALL  "FC892_Obtener_ValorDelAtributo"
      ( DB_String := #DBEventosRec,
        OffsetIni := #OffsetInicial,
        Valor     := #ValorDeAtributo
      );

      L     #ValorDeAtributo;  // Lo guardo
      T     #AtributosDeUTs.CotaAnchura;

// Continuo con el Evento
      L     #P_Eventos;
      LAR2;
      JU    InicioBucleAtributos_EventosDeLasUTs;



NETWORK
TITLE = ---- ---- Recoger el Atributo de las UTs - COTL (Cota de Profundidad)
/////////////////////////////////////////////////////////////////////////
/////////////////////////////////////////////////////////////////////////
/////////////////////////////////////////////////////////////////////////
AtributoDeUTs_COTL:NOP   0;
      +AR2  P#5.0;
      TAR2;
      T     #P_Eventos;
      SRD   3;
      T     #OffsetInicial;

// Obtener el Valor del Atributo
      CALL  "FC892_Obtener_ValorDelAtributo"
      ( DB_String := #DBEventosRec,
        OffsetIni := #OffsetInicial,
        Valor     := #ValorDeAtributo
      );

      L     #ValorDeAtributo;  // Lo guardo
      T     #AtributosDeUTs.CotaProfundidad;

// Continuo con el Evento
      L     #P_Eventos;
      LAR2;
      JU    InicioBucleAtributos_EventosDeLasUTs;



NETWORK
TITLE = ---- ---- Recoger el Atributo de las UTs - PESO
/////////////////////////////////////////////////////////////////////////
/////////////////////////////////////////////////////////////////////////
/////////////////////////////////////////////////////////////////////////
AtributoDeUTs_PESO:NOP   0;
      +AR2  P#5.0;
      TAR2;
      T     #P_Eventos;
      SRD   3;
      T     #OffsetInicial;

// Obtener el Valor del Atributo
      CALL  "FC892_Obtener_ValorDelAtributo"
      ( DB_String := #DBEventosRec,
        OffsetIni := #OffsetInicial,
        Valor     := #ValorDeAtributo
      );

      L     #ValorDeAtributo;  // Lo guardo
      T     #AtributosDeUTs.Peso;

// Continuo con el Evento
      L     #P_Eventos;
      LAR2;
      JU    InicioBucleAtributos_EventosDeLasUTs;



NETWORK
TITLE = ---- ---- Recoger el Atributo de las UTs - ALTO (Codigo de Altura)
/////////////////////////////////////////////////////////////////////////
/////////////////////////////////////////////////////////////////////////
/////////////////////////////////////////////////////////////////////////
AtributoDeUTs_ALTO:NOP   0;
      +AR2  P#5.0;
      TAR2;
      T     #P_Eventos;
      SRD   3;
      T     #OffsetInicial;

// Obtener el Valor del Atributo
      CALL  "FC892_Obtener_ValorDelAtributo"
      ( DB_String := #DBEventosRec,
        OffsetIni := #OffsetInicial,
        Valor     := #ValorDeAtributo
      );

      L     #ValorDeAtributo;  // Lo guardo
      T     #AtributosDeUTs.GaliboAltura;

// Continuo con el Evento
      L     #P_Eventos;
      LAR2;
      JU    InicioBucleAtributos_EventosDeLasUTs;



NETWORK
TITLE = ---- ---- Recoger el Atributo de las UTs - ANCH (Codigo de Anchura)
/////////////////////////////////////////////////////////////////////////
/////////////////////////////////////////////////////////////////////////
/////////////////////////////////////////////////////////////////////////
AtributoDeUTs_ANCH:NOP   0;
      +AR2  P#5.0;
      TAR2;
      T     #P_Eventos;
      SRD   3;
      T     #OffsetInicial;

// Obtener el Valor del Atributo
      CALL  "FC892_Obtener_ValorDelAtributo"
      ( DB_String := #DBEventosRec,
        OffsetIni := #OffsetInicial,
        Valor     := #ValorDeAtributo
      );

      L     #ValorDeAtributo;  // Lo guardo
      T     #AtributosDeUTs.GaliboAnchura;

// Continuo con el Evento
      L     #P_Eventos;
      LAR2;
      JU    InicioBucleAtributos_EventosDeLasUTs;



NETWORK
TITLE = ---- ---- Recoger el Atributo de las UTs - PROF (Codigo de Profundidad)
/////////////////////////////////////////////////////////////////////////
/////////////////////////////////////////////////////////////////////////
/////////////////////////////////////////////////////////////////////////
AtributoDeUTs_PROF:NOP   0;
      +AR2  P#5.0;
      TAR2;
      T     #P_Eventos;
      SRD   3;
      T     #OffsetInicial;

// Obtener el Valor del Atributo
      CALL  "FC892_Obtener_ValorDelAtributo"
      ( DB_String := #DBEventosRec,
        OffsetIni := #OffsetInicial,
        Valor     := #ValorDeAtributo
      );

      L     #ValorDeAtributo;  // Lo guardo
      T     #AtributosDeUTs.GaliboProfundidad;

// Continuo con el Evento
      L     #P_Eventos;
      LAR2;
      JU    InicioBucleAtributos_EventosDeLasUTs;



NETWORK
TITLE = ---- ---- Recoger el Atributo de las UTs - TACO (Codigo de Taco)
/////////////////////////////////////////////////////////////////////////
/////////////////////////////////////////////////////////////////////////
/////////////////////////////////////////////////////////////////////////
AtributoDeUTs_TACO:NOP   0;
      +AR2  P#5.0;
      TAR2;
      T     #P_Eventos;
      SRD   3;
      T     #OffsetInicial;

// Obtener el Valor del Atributo
      CALL  "FC892_Obtener_ValorDelAtributo"
      ( DB_String := #DBEventosRec,
        OffsetIni := #OffsetInicial,
        Valor     := #ValorDeAtributo
      );

      L     #ValorDeAtributo;  // Lo guardo
      T     #AtributosDeUTs.GaliboTaco;

// Continuo con el Evento
      L     #P_Eventos;
      LAR2;
      JU    InicioBucleAtributos_EventosDeLasUTs;



NETWORK
TITLE = ---- ---- Recoger el Atributo de las UTs - HUEC (Codigo de Hueco)
/////////////////////////////////////////////////////////////////////////
/////////////////////////////////////////////////////////////////////////
/////////////////////////////////////////////////////////////////////////
AtributoDeUTs_HUEC:NOP   0;
      +AR2  P#5.0;
      TAR2;
      T     #P_Eventos;
      SRD   3;
      T     #OffsetInicial;

// Obtener el Valor del Atributo
      CALL  "FC892_Obtener_ValorDelAtributo"
      ( DB_String := #DBEventosRec,
        OffsetIni := #OffsetInicial,
        Valor     := #ValorDeAtributo
      );

      L     #ValorDeAtributo;  // Lo guardo
      T     #AtributosDeUTs.GaliboHueco;

// Continuo con el Evento
      L     #P_Eventos;
      LAR2;
      JU    InicioBucleAtributos_EventosDeLasUTs;



NETWORK
TITLE = ---- ---- Recoger el Atributo de las UTs - HUER (Codigo de Hueco de Remontada)
/////////////////////////////////////////////////////////////////////////
/////////////////////////////////////////////////////////////////////////
/////////////////////////////////////////////////////////////////////////
AtributoDeUTs_HUER:NOP   0;
      +AR2  P#5.0;
      TAR2;
      T     #P_Eventos;
      SRD   3;
      T     #OffsetInicial;

// Obtener el Valor del Atributo
      CALL  "FC892_Obtener_ValorDelAtributo"
      ( DB_String := #DBEventosRec,
        OffsetIni := #OffsetInicial,
        Valor     := #ValorDeAtributo
      );

      L     #ValorDeAtributo;  // Lo guardo
      T     #AtributosDeUTs.GaliboHuecoRemontada;

// Continuo con el Evento
      L     #P_Eventos;
      LAR2;
      JU    InicioBucleAtributos_EventosDeLasUTs;



NETWORK
TITLE = ---- ---- Recoger el Atributo de las UTs - COLO (Codigo de Color)
/////////////////////////////////////////////////////////////////////////
/////////////////////////////////////////////////////////////////////////
/////////////////////////////////////////////////////////////////////////
AtributoDeUTs_COLO:NOP   0;
      +AR2  P#5.0;

      OPN   DB [#DBEventosRec];
      L     DBD [AR2, P#0.0];
      T     #EtiquetaAtributo;

// Obtener el Valor del Atributo
      CALL  "FC894_Obtener_ValorDeEtiqueta"
      ( EtiquetaEvento := #EtiquetaAtributo,
        ValorEvento    := #ValorDeEtiqueta
      );

      L     #ValorDeEtiqueta;  // Lo guardo
      T     #AtributosDeUTs.GaliboColor;

// Continuo con el Evento
      +AR2  P#4.0;
      JU    InicioBucleAtributos_EventosDeLasUTs;



NETWORK
TITLE = ---- ---- Recoger el Atributo de las UTs - PATI (Codigo de Patin)
/////////////////////////////////////////////////////////////////////////
/////////////////////////////////////////////////////////////////////////
/////////////////////////////////////////////////////////////////////////
AtributoDeUTs_PATI:NOP   0;
      +AR2  P#5.0;
      TAR2;
      T     #P_Eventos;
      SRD   3;
      T     #OffsetInicial;

// Obtener el Valor del Atributo
      CALL  "FC892_Obtener_ValorDelAtributo"
      ( DB_String := #DBEventosRec,
        OffsetIni := #OffsetInicial,
        Valor     := #ValorDeAtributo
      );

      L     #ValorDeAtributo;  // Lo guardo
      T     #AtributosDeUTs.GaliboPatin;

// Continuo con el Evento
      L     #P_Eventos;
      LAR2;
      JU    InicioBucleAtributos_EventosDeLasUTs;



NETWORK
TITLE = ---- ---- Recoger el Atributo de las UTs - LETI (Lado de la Etiqueta)
/////////////////////////////////////////////////////////////////////////
/////////////////////////////////////////////////////////////////////////
/////////////////////////////////////////////////////////////////////////
AtributoDeUTs_LETI:NOP   0;
      +AR2  P#5.0;
      TAR2;
      T     #P_Eventos;
      SRD   3;
      T     #OffsetInicial;

// Obtener el Valor del Atributo
      CALL  "FC892_Obtener_ValorDelAtributo"
      ( DB_String := #DBEventosRec,
        OffsetIni := #OffsetInicial,
        Valor     := #ValorDeAtributo
      );

      L     #ValorDeAtributo;  // Lo guardo
      L     1;
      +I;
      T     #AtributosDeUTs.PosicionDeLaEtiqueta;

// Continuo con el Evento
      L     #P_Eventos;
      LAR2;
      JU    InicioBucleAtributos_EventosDeLasUTs;



NETWORK
TITLE = ---- ---- Recoger el Atributo de las UTs - SGAP ( SGA - Error de Peso)
/////////////////////////////////////////////////////////////////////////
/////////////////////////////////////////////////////////////////////////
/////////////////////////////////////////////////////////////////////////
AtributoDeUTs_SGAP:NOP   0;
      +AR2  P#5.0;

      OPN   DB [#DBEventosRec];
      L     DBW [AR2, P#0.0];
      T     #Leido;

      L     0;  // Por defecto No Error
      T     #ValorDeAtributo;

      L     'NO';  // Tiene Error ?
      L     #Leido;
      ==I;
      JC    AtributoDeUTs_SGAP_NoError;

      L     W#16#08;
      T     #ValorDeAtributo;

AtributoDeUTs_SGAP_NoError:NOP   0;
      L     #ValorDeAtributo;
      L     #AtributosDeUTs.GaliboSGA;
      +I;
      T     #AtributosDeUTs.GaliboSGA;

// Continuo con el Evento
      +AR2  P#2.0;
      JU    InicioBucleAtributos_EventosDeLasUTs;



NETWORK
TITLE = ---- ---- Recoger el Atributo de las UTs - SGAE ( SGA - Error de Etiqueta)
/////////////////////////////////////////////////////////////////////////
/////////////////////////////////////////////////////////////////////////
/////////////////////////////////////////////////////////////////////////
AtributoDeUTs_SGAE:NOP   0;
      +AR2  P#5.0;

      OPN   DB [#DBEventosRec];
      L     DBW [AR2, P#0.0];
      T     #Leido;

      L     0;  // Por defecto No Error
      T     #ValorDeAtributo;

      L     'NO';  // Tiene Error ?
      L     #Leido;
      ==I;
      JC    AtributoDeUTs_SGAE_NoError;

      L     W#16#04;
      T     #ValorDeAtributo;

AtributoDeUTs_SGAE_NoError:NOP   0;
      L     #ValorDeAtributo;
      L     #AtributosDeUTs.GaliboSGA;
      +I;
      T     #AtributosDeUTs.GaliboSGA;

// Continuo con el Evento
      +AR2  P#2.0;
      JU    InicioBucleAtributos_EventosDeLasUTs;



NETWORK
TITLE = ---- ---- Recoger el Atributo de las UTs - SGAD ( SGA - Error de Dimensiones)
/////////////////////////////////////////////////////////////////////////
/////////////////////////////////////////////////////////////////////////
/////////////////////////////////////////////////////////////////////////
AtributoDeUTs_SGAD:NOP   0;
      +AR2  P#5.0;

      OPN   DB [#DBEventosRec];
      L     DBW [AR2, P#0.0];
      T     #Leido;

      L     0;  // Por defecto No Error
      T     #ValorDeAtributo;

      L     'NO';  // Tiene Error ?
      L     #Leido;
      ==I;
      JC    AtributoDeUTs_SGAD_NoError;

      L     W#16#02;
      T     #ValorDeAtributo;

AtributoDeUTs_SGAD_NoError:NOP   0;
      L     #ValorDeAtributo;
      L     #AtributosDeUTs.GaliboSGA;
      +I;
      T     #AtributosDeUTs.GaliboSGA;

// Continuo con el Evento
      +AR2  P#2.0;
      JU    InicioBucleAtributos_EventosDeLasUTs;



NETWORK
TITLE = ---- ---- Recoger el Atributo de las UTs - SGA_ ( SGA - Error General)
/////////////////////////////////////////////////////////////////////////
/////////////////////////////////////////////////////////////////////////
/////////////////////////////////////////////////////////////////////////
AtributoDeUTs_SGA_Error:NOP   0;
      +AR2  P#5.0;

      OPN   DB [#DBEventosRec];
      L     DBW [AR2, P#0.0];
      T     #Leido;

      L     0;  // Por defecto No Error
      T     #ValorDeAtributo;

      L     'NO';  // Tiene Error ?
      L     #Leido;
      ==I;
      JC    AtributoDeUTs_SGA_Error_NoError;

      L     W#16#01;
      T     #ValorDeAtributo;

AtributoDeUTs_SGA_Error_NoError:NOP   0;
      L     #ValorDeAtributo;
      L     #AtributosDeUTs.GaliboSGA;
      +I;
      T     #AtributosDeUTs.GaliboSGA;

// Continuo con el Evento
      +AR2  P#2.0;
      JU    InicioBucleAtributos_EventosDeLasUTs;



NETWORK
TITLE = ---- ---- Recoger el Atributo de las UTs - RSLT (Mover UT - Resultado)
/////////////////////////////////////////////////////////////////////////
/////////////////////////////////////////////////////////////////////////
/////////////////////////////////////////////////////////////////////////
AtributoDeUTs_RSLT:NOP   0;
      +AR2  P#5.0;

      OPN   DB [#DBEventosRec];
      L     DBW [AR2, P#0.0];  // Sacar el Valor del Campo
      T     #Leido;

      SET;  // Inicializar a NOK
      S     #AtributosDeUTs.CambiarUTDeMesa.NOK;
      R     #AtributosDeUTs.CambiarUTDeMesa.OK;

      L     #Leido;  // Comparar si es NO ?
      L     'SI';
      <>I;
      JC    InicioBucleAtributos_EventosDeLasUTs;

      SET;  // Inicializar a OK
      R     #AtributosDeUTs.CambiarUTDeMesa.NOK;
      S     #AtributosDeUTs.CambiarUTDeMesa.OK;

// Continuo con el Evento
      +AR2  P#2.0;
      JU    InicioBucleAtributos_EventosDeLasUTs;



NETWORK
TITLE = ---- ---- Recoger el Atributo de las UTs - PDST (Mover UT - Posicion en la Cola de Mesa)
/////////////////////////////////////////////////////////////////////////
/////////////////////////////////////////////////////////////////////////
/////////////////////////////////////////////////////////////////////////
AtributoDeUTs_PDST:NOP   0;
      +AR2  P#5.0;

      OPN   DB [#DBEventosRec];
      L     DBD [AR2, P#0.0];  // Sacar el Valor del Campo
      T     #EtiquetaAtributo;

      SET;  // Inicializar a Final
      S     #AtributosDeUTs.CambiarUTDeMesa.Final;
      R     #AtributosDeUTs.CambiarUTDeMesa.Inicio;

      L     #EtiquetaAtributo;  // Comparar si es _FIN ?
      L     '_INI';
      <>D;
      JC    InicioBucleAtributos_EventosDeLasUTs;

      SET;  // Inicializar a Inicio
      R     #AtributosDeUTs.CambiarUTDeMesa.Final;
      S     #AtributosDeUTs.CambiarUTDeMesa.Inicio;

// Continuo con el Evento
      +AR2  P#4.0;
      JU    InicioBucleAtributos_EventosDeLasUTs;



NETWORK
TITLE = ---- ---- Recoger el Atributo de las UTs - DEST (Mover UT - Destino)
/////////////////////////////////////////////////////////////////////////
/////////////////////////////////////////////////////////////////////////
/////////////////////////////////////////////////////////////////////////
AtributoDeUTs_DEST:NOP   0;
      +AR2  P#5.0;
      TAR2;
      T     #P_Eventos;
      SRD   3;
      T     #OffsetInicial;

// Obtener el Valor del Atributo
      CALL  "FC892_Obtener_ValorDelAtributo"
      ( DB_String := #DBEventosRec,
        OffsetIni := #OffsetInicial,
        Valor     := #ValorDeAtributo
      );

      L     #ValorDeAtributo;  // Lo guardo
      L     #AtributosDeUTs.CambiarUTDeMesa.Destino;

// Continuo con el Evento
      L     #P_Eventos;
      LAR2;
      JU    InicioBucleAtributos_EventosDeLasUTs;



NETWORK
TITLE = ////////////////////////////////////////////////////////////////////////////////////////////////////////////

NETWORK
TITLE = Analizar la lista de los Atributos de los Dispositivos
Atributos_EventosDeLosDispositivos:NOP   0;

/////////////////////////////////////////////////////////////////////////
/////////////////////////////////////////////////////////////////////////
/////////////////////////////////////////////////////////////////////////
// Inicializa variables de los Atributos de las UTs
      L     0;
      T     #Cero;

      CALL  FILL
      ( BVAL    := #Cero,
        RET_VAL := #ReturnValor,
        BLK     := #AtributosDeDispositivos
      );  // Inicializa Atributos de las UTS



NETWORK
TITLE = ----
/////////////////////////////////////////////////////////////////////////
/////////////////////////////////////////////////////////////////////////
// Buscando Atributos o Final del Evento
      +AR2  P#4.0;  // Prepara Puntero para ver los atributos

InicioBucleAtributos_EventosDeLosDispositivos:NOP   0;
      OPN   DB [#DBEventosRec];
      L     DBB [AR2, P#0.0];
      T     #Leido;

// Inicio de atributo - Ir a tratar los atributos
      L     #Leido;
      L     '[';  // '[' - Inicio de Atributo
      ==I;  // Atributo del Evento
      JC    EncontradoAtributos_EventosDeLosDispositivos;

// Fin del Evento
      L     #Leido;
      L     '}';  // '}' - Fin del Evento
      ==I;  // Se acabo el evento
      JC    FinalAtributos_EventosDeLosDispositivos;

      +AR2  P#1.0;  // Seguir buscado atributo
      JU    InicioBucleAtributos_EventosDeLosDispositivos;


/////////////////////////////////////////////////////////////////////////
/////////////////////////////////////////////////////////////////////////
// Se acaba el Evento - Ir a guardar datos del Evento
FinalAtributos_EventosDeLosDispositivos:NOP   0;
      TAR2;
      T     #P_Eventos;  // Guardo Por donde voy en la lista de eventos
      JU    GuardarDatos_EventosRecibidos;



NETWORK
TITLE = Distribucion de los Atributos de los DIspositivos (LIsta del DB de Conversion)
EncontradoAtributos_EventosDeLosDispositivos:NOP   0;

/////////////////////////////////////////////////////////////////////////
/////////////////////////////////////////////////////////////////////////
/////////////////////////////////////////////////////////////////////////
/////////////////////////////////////////////////////////////////////////
// Mirar que Atributo del Evento  es ?
      +AR2  P#1.0;
      OPN   DB [#DBEventosRec];
      L     DBD [AR2, P#0.0];  // Atributo - 4 Caracteres
      T     #Atributo;

/////////////////////////////////////////////////////////////////////////
/////////////////////////////////////////////////////////////////////////
/////////////////////////////////////////////////////////////////////////
// Buscar numero de Atributo
      L     1;
      T     #NumeroAtributo;
BucleDeBusqueda_NumeroDeAtributoDeDispositivos:NOP   0;

// -- Se ha encontrado el Atributo Recibido
      L     "DB870_ConversorEventos".AtributosRecibidosDeDispositivos[#NumeroAtributo];
      L     #Atributo;
      ==D;
      JC    Encontrado_NumeroDeAtributoDeDispositivos;

// -- Final de la lista de Atributo Recibidos - No Encontrado
      L     "DB870_ConversorEventos".AtributosRecibidosDeDispositivos[#NumeroAtributo];
      L     0;
      ==D;
      JC    InicioBucleAtributos_EventosDeLosDispositivos;

// --- Maximo del Array de la Lista de Atributo Recibidos - No Encontrado
      L     #NumeroAtributo;
      L     "CTE_MaxArrayConversion";
      >=I;
      JC    InicioBucleAtributos_EventosDeLosDispositivos;


// --- Continuar la Busqueda
      L     #NumeroAtributo;
      L     1;
      +I;
      T     #NumeroAtributo;
      JU    BucleDeBusqueda_NumeroDeAtributoDeDispositivos;



NETWORK
TITLE = ----
/////////////////////////////////////////////////////////////////////////
/////////////////////////////////////////////////////////////////////////
/////////////////////////////////////////////////////////////////////////
// Distribuir dependiendo del Resultado de la Busqueda de Atributo Recibido
Encontrado_NumeroDeAtributoDeDispositivos:NOP   0;
      L     #NumeroAtributo;
      JL    NoExiste_NumeroDeAtibutoDeDispositivos;

      JU    NoExiste_NumeroDeAtibutoDeDispositivos;
      JU    AtributoDeDispositivos_TIPO;  // Atributo (01) - TIPO
      JU    AtributoDeDispositivos_NUME;  // Atributo (02) - NUME
      JU    AtributoDeDispositivos_NUES;  // Atributo (03) - NUES
      JU    AtributoDeDispositivos_HABI;  // Atributo (04) - HABI
      JU    AtributoDeDispositivos_PRIO;  // Atributo (05) - PRIO

      JU    AtributoDeDispositivos_SONO;  // Atributo (06) - SONO
      JU    AtributoDeDispositivos_VERD;  // Atributo (07) - VERD
      JU    AtributoDeDispositivos_ROJO;  // Atributo (08) - ROJO
      JU    AtributoDeDispositivos_AMAR;  // Atributo (09) - AMAR
      JU    AtributoDeDispositivos_AZUL;  // Atributo (10) - AZUL

      JU    AtributoDeDispositivos_MOTI;  // Atributo (11) - MOTI
      JU    AtributoDeDispositivos_OPER;  // Atributo (12) - OPER
      JU    AtributoDeDispositivos_TEXT;  // Atributo (13) - TEXT

      JU    AtributoDeDispositivos_HORQ;  // Atributo (14) - HORQ
      JU    AtributoDeDispositivos_POSI;  // Atributo (15) - POSI

/////////////////////////////////////////////////////////////////////////
NoExiste_NumeroDeAtibutoDeDispositivos:NOP   0;
      JU    InicioBucleAtributos_EventosDeLosDispositivos;



NETWORK
TITLE = ---- ---- Recoger el Atributo de los Dispositivos - TIPO
/////////////////////////////////////////////////////////////////////////
/////////////////////////////////////////////////////////////////////////
/////////////////////////////////////////////////////////////////////////
AtributoDeDispositivos_TIPO:NOP   0;
      +AR2  P#5.0;

      OPN   DB [#DBEventosRec];
      L     DBD [AR2, P#0.0];
      T     #EtiquetaAtributo;

// Obtener el Valor del Tipo de Dispositivo

      CALL  "FC894_Obtener_ValorDeEtiqueta"
      ( EtiquetaEvento := #EtiquetaAtributo,
        ValorEvento    := #ValorDeEtiqueta
      );

      L     #ValorDeEtiqueta;  // Lo guardo
      T     #AtributosDeDispositivos.Tipo;

// Continuo con el Evento
      +AR2  P#4.0;
      JU    InicioBucleAtributos_EventosDeLosDispositivos;



NETWORK
TITLE = ---- ---- Recoger el Atributo de los Dispositivos - NUME
/////////////////////////////////////////////////////////////////////////
/////////////////////////////////////////////////////////////////////////
/////////////////////////////////////////////////////////////////////////
AtributoDeDispositivos_NUME:NOP   0;
      +AR2  P#5.0;
      TAR2;
      T     #P_Eventos;
      SRD   3;
      T     #OffsetInicial;

// Obtener el Valor del Numero del Dispositivo

      CALL  "FC892_Obtener_ValorDelAtributo"
      ( DB_String := #DBEventosRec,
        OffsetIni := #OffsetInicial,
        Valor     := #ValorDeAtributo
      );
      L     #ValorDeAtributo;  // Lo guardo
      T     #AtributosDeDispositivos.Numero;

// Continuo con el Evento
      L     #P_Eventos;
      LAR2;
      JU    InicioBucleAtributos_EventosDeLosDispositivos;



NETWORK
TITLE = ---- ---- Recoger el Atributo de los Dispositivos - NUES (Nuevo Estado)
/////////////////////////////////////////////////////////////////////////
/////////////////////////////////////////////////////////////////////////
/////////////////////////////////////////////////////////////////////////
AtributoDeDispositivos_NUES:NOP   0;
      +AR2  P#5.0;

      OPN   DB [#DBEventosRec];
      L     DBD [AR2, P#0.0];
      T     #EtiquetaAtributo;

// Obtener el Valor del Tipo de Dispositivo
      CALL  "FC894_Obtener_ValorDeEtiqueta"
      ( EtiquetaEvento := #EtiquetaAtributo,
        ValorEvento    := #ValorDeEtiqueta
      );

      L     #ValorDeEtiqueta;  // Lo guardo
      T     #AtributosDeDispositivos.NuevoEstado;

// Continuo con el Evento
      +AR2  P#4.0;
      JU    InicioBucleAtributos_EventosDeLosDispositivos;



NETWORK
TITLE = ---- ---- Recoger el Atributo de los Dispositivos - HABI
/////////////////////////////////////////////////////////////////////////
/////////////////////////////////////////////////////////////////////////
/////////////////////////////////////////////////////////////////////////
AtributoDeDispositivos_HABI:NOP   0;
      +AR2  P#5.0;

      OPN   DB [#DBEventosRec];
      L     DBW [AR2, P#0.0];
      T     #Leido;

      L     2001;
      T     #ValorDeAtributo;

      L     #Leido;
      L     'NO';
      ==I;
      JCN   AtributoDeDispositivos_HABI_NoHabilitar;

      L     2002;
      T     #ValorDeAtributo;

AtributoDeDispositivos_HABI_NoHabilitar:NOP   0;
      L     #ValorDeAtributo;  // Lo guardo
      T     #AtributosDeDispositivos.Habilitado;

// Continuo con el Evento
      +AR2  P#2.0;
      JU    InicioBucleAtributos_EventosDeLosDispositivos;



NETWORK
TITLE = ---- ---- Recoger el Atributo de los Dispositivos - PRIO
/////////////////////////////////////////////////////////////////////////
/////////////////////////////////////////////////////////////////////////
/////////////////////////////////////////////////////////////////////////
AtributoDeDispositivos_PRIO:NOP   0;
      +AR2  P#5.0;
      TAR2;
      T     #P_Eventos;
      SRD   3;
      T     #OffsetInicial;

// Obtener el Valor del Numero del Dispositivo
      CALL  "FC892_Obtener_ValorDelAtributo"
      ( DB_String := #DBEventosRec,
        OffsetIni := #OffsetInicial,
        Valor     := #ValorDeAtributo
      );

      L     #ValorDeAtributo;  // Lo guardo
      L     1;
      +I;
      T     #AtributosDeDispositivos.Prioridad;

// Continuo con el Evento
      L     #P_Eventos;
      LAR2;
      JU    InicioBucleAtributos_EventosDeLosDispositivos;



NETWORK
TITLE = ---- ---- Recoger el Atributo de los Dispositivos - SONO (Baliza - Sirena)
/////////////////////////////////////////////////////////////////////////
/////////////////////////////////////////////////////////////////////////
/////////////////////////////////////////////////////////////////////////
AtributoDeDispositivos_SONO:NOP   0;
      +AR2  P#5.0;

      SET;
      S     #AtributosDeDispositivos.BalizaColor.Sonoro;


// Continuo con el Evento
      JU    InicioBucleAtributos_EventosDeLosDispositivos;



NETWORK
TITLE = ---- ---- Recoger el Atributo de los Dispositivos - VERD (Baliza - Verde)
/////////////////////////////////////////////////////////////////////////
/////////////////////////////////////////////////////////////////////////
/////////////////////////////////////////////////////////////////////////
AtributoDeDispositivos_VERD:NOP   0;
      +AR2  P#5.0;

      SET;
      S     #AtributosDeDispositivos.BalizaColor.Verde;


// Continuo con el Evento
      JU    InicioBucleAtributos_EventosDeLosDispositivos;



NETWORK
TITLE = ---- ---- Recoger el Atributo de los Dispositivos - ROJO (Baliza - Roja)
/////////////////////////////////////////////////////////////////////////
/////////////////////////////////////////////////////////////////////////
/////////////////////////////////////////////////////////////////////////
AtributoDeDispositivos_ROJO:NOP   0;
      +AR2  P#5.0;

      SET;
      S     #AtributosDeDispositivos.BalizaColor.Rojo;


// Continuo con el Evento
      JU    InicioBucleAtributos_EventosDeLosDispositivos;



NETWORK
TITLE = ---- ---- Recoger el Atributo de los Dispositivos - AMAR (Baliza - Amarilla)
/////////////////////////////////////////////////////////////////////////
/////////////////////////////////////////////////////////////////////////
/////////////////////////////////////////////////////////////////////////
AtributoDeDispositivos_AMAR:NOP   0;
      +AR2  P#5.0;

      SET;
      S     #AtributosDeDispositivos.BalizaColor.Amarillo;


// Continuo con el Evento
      JU    InicioBucleAtributos_EventosDeLosDispositivos;



NETWORK
TITLE = ---- ---- Recoger el Atributo de los Dispositivos - AZUL (Baliza - Azul)
/////////////////////////////////////////////////////////////////////////
/////////////////////////////////////////////////////////////////////////
/////////////////////////////////////////////////////////////////////////
AtributoDeDispositivos_AZUL:NOP   0;
      +AR2  P#5.0;

      SET;
      S     #AtributosDeDispositivos.BalizaColor.Azul;


// Continuo con el Evento
      JU    InicioBucleAtributos_EventosDeLosDispositivos;



NETWORK
TITLE = ---- ---- Recoger el Atributo de los Dispositivos - MOTI (Moitvo del Envio a Error del JdT )
/////////////////////////////////////////////////////////////////////////
/////////////////////////////////////////////////////////////////////////
/////////////////////////////////////////////////////////////////////////
AtributoDeDispositivos_MOTI:NOP   0;
      +AR2  P#5.0;

// - Recorrer el Motivo del Error es una STRING
      L     2;  // Inicializaciones
      T     #LonguitudTextoRecibido;

// Inicio a Recoger el Motivo del Error
AtributoDeDispositivos_MOTI_InicioBucle:NOP   0;
      OPN   DB [#DBEventosRec];
      L     DBB [AR2, P#0.0];  // Leer ek texto
      T     #Leido;

      L     #Leido;  // Es final del Texto
      L     '[';
      ==I;
      JC    AtributoDeDispositivos_MOTI_FinalBucle;

      L     #Leido;  // Es final del Texto
      L     '}';
      ==I;
      JC    AtributoDeDispositivos_MOTI_FinalBucle;

      L     #Leido;  // Guardo el texto
      T     #AtributosDeDispositivos.MotivoDelError[#LonguitudTextoRecibido];

// Incremetar punteros
      +AR2  P#1.0;
      L     #LonguitudTextoRecibido;
      L     1;
      +I;
      T     #LonguitudTextoRecibido;

      L     0;  // Pongo el siguiente a cero
      T     #AtributosDeDispositivos.MotivoDelError[#LonguitudTextoRecibido];

      JU    AtributoDeDispositivos_MOTI_InicioBucle;


// - Continuo con el Evento
AtributoDeDispositivos_MOTI_FinalBucle:NOP   0;
      L     48;  // Inicio la carcacteristica de la STRING
      T     #AtributosDeDispositivos.MotivoDelError[0];
      L     #LonguitudTextoRecibido;
      L     2;
      -I;
      T     #AtributosDeDispositivos.MotivoDelError[1];

      JU    InicioBucleAtributos_EventosDeLosDispositivos;



NETWORK
TITLE = ---- ---- Recoger el Atributo de los Dispositivos - OPER (Operacion a realizar de las Maquinas)
/////////////////////////////////////////////////////////////////////////
/////////////////////////////////////////////////////////////////////////
/////////////////////////////////////////////////////////////////////////
AtributoDeDispositivos_OPER:NOP   0;
      +AR2  P#5.0;

      OPN   DB [#DBEventosRec];
      L     DBD [AR2, P#0.0];
      T     #EtiquetaAtributo;

// Obtener el Valor del Tipo de Dispositivo
      CALL  "FC894_Obtener_ValorDeEtiqueta"
      ( EtiquetaEvento := #EtiquetaAtributo,
        ValorEvento    := #ValorDeEtiqueta
      );

      L     #ValorDeEtiqueta;  // Lo guardo
      T     #AtributosDeDispositivos.Operacion;

// Continuo con el Evento
      +AR2  P#4.0;
      JU    InicioBucleAtributos_EventosDeLosDispositivos;



NETWORK
TITLE = ---- ---- Recoger el Atributo de los Dispositivos - TEXT
/////////////////////////////////////////////////////////////////////////
/////////////////////////////////////////////////////////////////////////
/////////////////////////////////////////////////////////////////////////
AtributoDeDispositivos_TEXT:NOP   0;
      +AR2  P#5.0;

// - Recorrer el Motivo del Error es una STRING
      L     2;  // Inicializaciones
      T     #LonguitudTextoRecibido;

// Inicio a Recoger el Texto
AtributoDeDispositivos_TEXT_InicioBucle:NOP   0;
      OPN   DB [#DBEventosRec];
      L     DBB [AR2, P#0.0];  // Leer ek texto
      T     #Leido;

      L     #Leido;  // Es final del Texto
      L     '[';
      ==I;
      JC    AtributoDeDispositivos_TEXT_FinalBucle;

      L     #Leido;  // Es final del Texto
      L     '}';
      ==I;
      JC    AtributoDeDispositivos_TEXT_FinalBucle;

      L     #Leido;  // Guardo el texto
      T     #AtributosDeDispositivos.TextoRecibido[#LonguitudTextoRecibido];

// Incremetar punteros
      +AR2  P#1.0;
      L     #LonguitudTextoRecibido;
      L     1;
      +I;
      T     #LonguitudTextoRecibido;

      L     0;  // Pongo el siguiente a cero
      T     #AtributosDeDispositivos.TextoRecibido[#LonguitudTextoRecibido];

      JU    AtributoDeDispositivos_TEXT_InicioBucle;


// - Continuo con el Evento
AtributoDeDispositivos_TEXT_FinalBucle:NOP   0;
      L     48;  // Inicio la carcacteristica de la STRING
      T     #AtributosDeDispositivos.TextoRecibido[0];
      L     #LonguitudTextoRecibido;
      L     2;
      -I;
      T     #AtributosDeDispositivos.TextoRecibido[1];

      JU    InicioBucleAtributos_EventosDeLosDispositivos;



NETWORK
TITLE = ---- ---- Recoger el Atributo de los Dispositivos - HORQ
/////////////////////////////////////////////////////////////////////////
/////////////////////////////////////////////////////////////////////////
/////////////////////////////////////////////////////////////////////////
AtributoDeDispositivos_HORQ:NOP   0;
      +AR2  P#5.0;
      TAR2;
      T     #P_Eventos;
      SRD   3;
      T     #OffsetInicial;

// Obtener el Valor del Numero del Dispositivo
      CALL  "FC892_Obtener_ValorDelAtributo"
      ( DB_String := #DBEventosRec,
        OffsetIni := #OffsetInicial,
        Valor     := #ValorDeAtributo
      );
      L     #ValorDeAtributo;  // Lo guardo
      T     #AtributosDeDispositivos.MesaHorquilla;

// Continuo con el Evento
      L     #P_Eventos;
      LAR2;
      JU    InicioBucleAtributos_EventosDeLosDispositivos;



NETWORK
TITLE = ---- ---- Recoger el Atributo de los Dispositivos - POSI
/////////////////////////////////////////////////////////////////////////
/////////////////////////////////////////////////////////////////////////
/////////////////////////////////////////////////////////////////////////
AtributoDeDispositivos_POSI:NOP   0;
      +AR2  P#5.0;
      TAR2;
      T     #P_Eventos;
      SRD   3;
      T     #OffsetInicial;

// Obtener el Valor del Numero del Dispositivo
      CALL  "FC892_Obtener_ValorDelAtributo"
      ( DB_String := #DBEventosRec,
        OffsetIni := #OffsetInicial,
        Valor     := #ValorDeAtributo
      );
      L     #ValorDeAtributo;  // Lo guardo
      T     #AtributosDeDispositivos.MesaCargaDesCarga;

// Continuo con el Evento
      L     #P_Eventos;
      LAR2;
      JU    InicioBucleAtributos_EventosDeLosDispositivos;



NETWORK
TITLE = Distribucion para Guardar Datos del Evento Recibido (LIsta del DB de Conversion) ///////
/////////////////////////////////////////////////////////////////////////
/////////////////////////////////////////////////////////////////////////
/////////////////////////////////////////////////////////////////////////
GuardarDatos_EventosRecibidos:NOP   0;
      TAR2;
      T     #P_Eventos;  // Guardo Por donde voy en la lista de eventos

      L     #NumeroEvento;
      JL    NoExiste_GuardarDatos_Eventos;

      JU    NoExiste_GuardarDatos_Eventos;
      JU    GuardarDatos_EventoRecibido_CREA;  // Evento (01) - CREA
      JU    GuardarDatos_EventoRecibido_RUTA;  // Evento (02) - RUTA
      JU    GuardarDatos_EventoRecibido_DRUT;  // Evento (03) - DRUT
      JU    GuardarDatos_EventoRecibido_RETI;  // Evento (04) - RETI
      JU    GuardarDatos_EventoRecibido_BORR;  // Evento (05) - BORR
      JU    GuardarDatos_EventoRecibido_DATA;  // Evento (06) - DATA
      JU    GuardarDatos_EventoRecibido_Refresco_UT;  // Evento (07) - ?UT?
      JU    GuardarDatos_EventoRecibido_MOVE;  // Evento (08) - MOVE
      JU    GuardarDatos_EventoRecibido_DEMB;  // Evento (09) - DEMB

      JU    GuardarDatos_EventoRecibido_CSTA;  // Evento (10) - CSTA
      JU    GuardarDatos_EventoRecibido_DIDO;  // Evento (11) - DIDO

      JU    NoExiste_GuardarDatos_Eventos;  // Evento (12) - ORDE
      JU    NoExiste_GuardarDatos_Eventos;  // Evento (13) - BOET
      JU    NoExiste_GuardarDatos_Eventos;  // Evento (14) - BOBD
      JU    NoExiste_GuardarDatos_Eventos;  // Evento (15) - RUET
      JU    NoExiste_GuardarDatos_Eventos;  // Evento (16) - RUES
      JU    NoExiste_GuardarDatos_Eventos;  // Evento (17) - INIR

      JU    GuardarDatos_EventoRecibido_Refresco_ST;  // Evento (18) - ?ST?

      JU    NoExiste_GuardarDatos_Eventos;  // Evento (19) - QCRE
      JU    NoExiste_GuardarDatos_Eventos;  // Evento (20) - QPR?

      JU    NoExiste_GuardarDatos_Eventos;  // Evento (21) - CHEQ

/////////////////////////////////////////////////////////////////////////
NoExiste_GuardarDatos_Eventos:NOP   0;
      L     #P_Eventos;  // Recupero por donde voy en la lista de eventos
      LAR2;  // Regreso a buscar el siguiente evento
      JU    FinBucle_EventosRecibidos;



NETWORK
TITLE = ////////////////////////////////////////////////////////////////////////////////////////////////////////////

NETWORK
TITLE = Guardar Datos - Evento CREA - Crear una Nueva UT
// Analisis del evento
//   - Inicializa variables de los atributos del Evento
//   - Buscar Atributos o Final del Evento
//   - Guardar datos del Evento
// Analisis de los atributos del Evento
//   - Mirar que atributo del Evento es
//   - Distribuir a recoger los datos del Evento
//   - Recoger el Atributo McKey
//   - Recoger el Atributo MesaActual
//   - Recoger el Atributo Tipo
//   - Recoger el Atributo Codigo de Barras
//   - Recoger el Atributo Grupo de UT
//   - Recoger el Atributo Cantidad de UT en el Grupo
//   - Recoger el Atributo Orden dentro del grupo
//   - Recoger el Atributo Altura
GuardarDatos_EventoRecibido_CREA:NOP   0;

/////////////////////////////////////////////////////////////////////////
/////////////////////////////////////////////////////////////////////////
/////////////////////////////////////////////////////////////////////////
// --- Guardar Datos del Evento Recibido


/////////////////////////////////////////////////////////////////////////
/////////////////////////////////////////////////////////////////////////
/////////////////////////////////////////////////////////////////////////
// --- Control de la Mesa Actual es correcta
      L     #AtributosDeUTs.MesaActual;  // Ver que mesa es
      L     "CTE_OffsetMesa";
      -I;
      T     #VarTempUTs.MesaActual;

      L     #VarTempUTs.MesaActual;  // Comprobar el numero de mesa
      L     1;  // No menor de 1
      <I;  // No es correcto
      JC    Final_EventoRecibido_CREA;
      L     #VarTempUTs.MesaActual;
      L     "CTE_MaxMesas";  // No mayor que el parametro
      >I;  // No es correcto
      JC    Final_EventoRecibido_CREA;


/////////////////////////////////////////////////////////////////////////
/////////////////////////////////////////////////////////////////////////
/////////////////////////////////////////////////////////////////////////
// --- Control del Mckey es correcto
      L     #AtributosDeUTs.Mckey;  // Se ha recibido Mckey = 0
      L     0;  // No se puede Crear
      ==D;
      JC    Final_EventoRecibido_CREA;


/////////////////////////////////////////////////////////////////////////
/////////////////////////////////////////////////////////////////////////
/////////////////////////////////////////////////////////////////////////
// --- Control del Nuevo Mckey no este en el sistema
// --- Comprobación de DUPLICIDAD
      CALL  "FC720_BuscarUT_EnMesa"
      ( Mckey      := #AtributosDeUTs.Mckey,
        MesaActual := #VarTempUTs.MesaActual,
        NumeroUT   := #VarTempUTs.NumeroUT
      );

      L     #VarTempUTs.NumeroUT;  // Existe UT, Hay DUPLICIDAD de Mckey
      L     0;
      ==I;
      JC    MckeyCorrecto_EventoRecibido_CREA;

// --- Informe de Duplicadad del Mckey
      SET;
      S     "DB812_UTs_Control".UT[#VarTempUTs.NumeroUT].EventosInformarJdT.DuplicidadMckey;

      JU    Final_EventoRecibido_CREA;

MckeyCorrecto_EventoRecibido_CREA:NOP   0;


/////////////////////////////////////////////////////////////////////////
/////////////////////////////////////////////////////////////////////////
/////////////////////////////////////////////////////////////////////////
// --- Control de la Mesa este Definida
      SET;
      AN    "DB850_DefinicionMesas".Mesa[#VarTempUTs.MesaActual].ConfigMesa.MesaPaso;
      AN    "DB850_DefinicionMesas".Mesa[#VarTempUTs.MesaActual].ConfigMesa.MesaCruce;
      AN    "DB850_DefinicionMesas".Mesa[#VarTempUTs.MesaActual].ConfigMesa.MesaMultiplesDestinos;
      JC    Final_EventoRecibido_CREA;


/////////////////////////////////////////////////////////////////////////
/////////////////////////////////////////////////////////////////////////
/////////////////////////////////////////////////////////////////////////
// --- Crear UT en la Mesa Actual
// --- Nota: Rellena ya en UT el Mckey y la Mesa Actual
      CALL  "FC721_CrearUT_EnMesa"
      ( McKey      := #AtributosDeUTs.Mckey,
        MesaActual := #VarTempUTs.MesaActual,
        NumeroUT   := #VarTempUTs.NumeroUT
      );

      L     #VarTempUTs.NumeroUT;
      L     0;  // No se ha podido crear
      ==I;
      JC    Final_EventoRecibido_CREA;



NETWORK
TITLE = ---- Accion del Evento
/////////////////////////////////////////////////////////////////////////
/////////////////////////////////////////////////////////////////////////
/////////////////////////////////////////////////////////////////////////
// --- Guardar datos en la UT, Mckey y Mesa ya estan
      L     202;  // 202 - Recibido Evento de Creada una Nueva UT en la Mesa
      T     "DB812_UTs_Control".UT[#VarTempUTs.NumeroUT].EstadoEventoRecibido;

      L     #AtributosDeUTs.TipoCarga;
      T     "DB812_UTs_Control".UT[#VarTempUTs.NumeroUT].TipoCarga;

      SET;
      A     #AtributosDeUTs.AtributosTipoDeCarga.Pila;
      S     "DB812_UTs_Control".UT[#VarTempUTs.NumeroUT].AtributosDelaCarga.Pila;
      SET;
      A     #AtributosDeUTs.AtributosTipoDeCarga.Remontada;
      S     "DB812_UTs_Control".UT[#VarTempUTs.NumeroUT].AtributosDelaCarga.Remontada;
      SET;
      A     #AtributosDeUTs.AtributosTipoDeCarga.Vacia;
      S     "DB812_UTs_Control".UT[#VarTempUTs.NumeroUT].AtributosDelaCarga.Vacia;


      L     #AtributosDeUTs.GaliboAltura;
      T     "DB815_UTs_Datos".UT[#VarTempUTs.NumeroUT].GaliboAltura;
      L     #AtributosDeUTs.GaliboAnchura;
      T     "DB815_UTs_Datos".UT[#VarTempUTs.NumeroUT].GaliboAnchura;
      L     #AtributosDeUTs.GaliboProfundidad;
      T     "DB815_UTs_Datos".UT[#VarTempUTs.NumeroUT].GaliboProfundidad;

      L     #AtributosDeUTs.GaliboTaco;
      T     "DB815_UTs_Datos".UT[#VarTempUTs.NumeroUT].GaliboTaco;
      L     #AtributosDeUTs.GaliboHueco;
      T     "DB815_UTs_Datos".UT[#VarTempUTs.NumeroUT].GaliboHueco;
      L     #AtributosDeUTs.GaliboHuecoRemontada;
      T     "DB815_UTs_Datos".UT[#VarTempUTs.NumeroUT].GaliboHuecoRemontado;

      L     #AtributosDeUTs.GaliboColor;
      T     "DB815_UTs_Datos".UT[#VarTempUTs.NumeroUT].GaliboColor;
      L     #AtributosDeUTs.GaliboPatin;
      T     "DB815_UTs_Datos".UT[#VarTempUTs.NumeroUT].GaliboPatin;


      L     #AtributosDeUTs.CodigoFlejado;
      T     "DB815_UTs_Datos".UT[#VarTempUTs.NumeroUT].CodigoFlejado;
      L     #AtributosDeUTs.CodigoEnfardado;
      T     "DB815_UTs_Datos".UT[#VarTempUTs.NumeroUT].CodigoEnfardado;
      L     #AtributosDeUTs.CodigoEtiquetado;
      T     "DB815_UTs_Datos".UT[#VarTempUTs.NumeroUT].CodigoEtiquetado;

      L     #AtributosDeUTs.Peso;
      T     "DB815_UTs_Datos".UT[#VarTempUTs.NumeroUT].Peso;

      L     #AtributosDeUTs.CotaAltura;
      T     "DB815_UTs_Datos".UT[#VarTempUTs.NumeroUT].CotaAltura;
      L     #AtributosDeUTs.CotaAnchura;
      T     "DB815_UTs_Datos".UT[#VarTempUTs.NumeroUT].CotaAnchura;
      L     #AtributosDeUTs.CotaProfundidad;
      T     "DB815_UTs_Datos".UT[#VarTempUTs.NumeroUT].CotaProfundidad;

      L     #AtributosDeUTs.CotaAmarre;
      T     "DB815_UTs_Datos".UT[#VarTempUTs.NumeroUT].Amarre;
      L     #AtributosDeUTs.Presion;
      T     "DB815_UTs_Datos".UT[#VarTempUTs.NumeroUT].Presion;

      L     #AtributosDeUTs.Grupo;
      T     "DB812_UTs_Control".UT[#VarTempUTs.NumeroUT].Grupo;
      L     #AtributosDeUTs.CantidadGrupo;
      T     "DB812_UTs_Control".UT[#VarTempUTs.NumeroUT].CantidadGrupo;
      L     #AtributosDeUTs.PosicionGrupo;
      T     "DB812_UTs_Control".UT[#VarTempUTs.NumeroUT].PosicionGrupo;


/////////////////////////////////////////////////////////////////////////
// --- Posicion de la Etiqueta (0) Derecha (1) Izquierdo
      SET;  // Posicion de la Etiqueta
      L     #AtributosDeUTs.PosicionDeLaEtiqueta;
      L     1;  // Lado Derecho = 0
      ==I;
      R     "DB812_UTs_Control".UT[#VarTempUTs.NumeroUT].AtributosDeLaUT.LadoDeLaEtiqueta;

      SET;  // Posicion de la Etiqueta
      L     #AtributosDeUTs.PosicionDeLaEtiqueta;
      L     2;  // Lado Izquierdo = 1
      ==I;
      S     "DB812_UTs_Control".UT[#VarTempUTs.NumeroUT].AtributosDeLaUT.LadoDeLaEtiqueta;


/////////////////////////////////////////////////////////////////////////
// --- Guardar la etiqueta
      CALL  BLKMOV
      ( SRCBLK  := #AtributosDeUTs.Etiqueta,
        RET_VAL := #ReturnValor,
        DSTBLK  := "DB814_UTs_Etiqueta".UT[#VarTempUTs.NumeroUT].Etiqueta
      );

/////////////////////////////////////////////////////////////////////////
// --- Guardar Datos de QUBIQA
      L     #AtributosDeUTs.QUBIQA_NumeroBulto;  // Numero de Bulto
      T     "DB820_UTs_DatosQUBIQA".UT[#VarTempUTs.NumeroUT].NumeroDeBulto;
      L     #AtributosDeUTs.QUBIQA_TotalBultos;  // Numero de Bultos
      T     "DB820_UTs_DatosQUBIQA".UT[#VarTempUTs.NumeroUT].TotalBultos;

      CALL  BLKMOV
      ( SRCBLK  := #AtributosDeUTs.QUBIQA_PID,
        RET_VAL := #ReturnValor,
        DSTBLK  := "DB820_UTs_DatosQUBIQA".UT[#VarTempUTs.NumeroUT].PID
      );  // Guardar el PID


/////////////////////////////////////////////////////////////////////////
// Guardar Ruta si es necesario
// Si hay ruta Nueva - Guardar MesaDestino, Mesa Intermedia y la nueva ruta
      L     0;  // Si existe Nueva Ruta - MesaDestino <> 0
      L     #AtributosDeUTs.MesaDestino;
      ==I;
      JC    FinalGuardarRuta_EventoRecibido_CREA;


/////////////////////////////////////////////////////////////////////////
// Puntero a la UT, Marcar si es necesario -->
//           Actual = Destino = InterMedia --> Marcar la UT
// MODIFICACION --> 06/05/2013 (Alonso)

      SET;  // Reset - Recircular la Carga - Memoria del Retirar
      R     "DB812_UTs_Control".UT[#VarTempUTs.NumeroUT].AtributosDeLaUT.RecircularCarga;
      R     "DB812_UTs_Control".UT[#VarTempUTs.NumeroUT].AtributosDeLaUT.MemorizarRETI;

      L     "DB812_UTs_Control".UT[#VarTempUTs.NumeroUT].MesaActual;
      L     #AtributosDeUTs.MesaDestino;
      <>I;  // MesaActual <> MesaDestino ?
      JC    NoRecirculaLaCarga_EventoRecibido_CREA;

      L     #AtributosDeUTs.MesaDestino;
      L     #AtributosDeUTs.Ruta[0];
      ==I;
      JC    NoRecirculaLaCarga_EventoRecibido_CREA;

      SET;  // Set - Recircular la Carga
      S     "DB812_UTs_Control".UT[#VarTempUTs.NumeroUT].AtributosDeLaUT.RecircularCarga;

NoRecirculaLaCarga_EventoRecibido_CREA:NOP   0;

      L     #AtributosDeUTs.MesaDestino;
      T     "DB812_UTs_Control".UT[#VarTempUTs.NumeroUT].MesaDestino;
      L     #AtributosDeUTs.MesaIntermedia;
      T     "DB812_UTs_Control".UT[#VarTempUTs.NumeroUT].MesaIntermedia;

      CALL  BLKMOV
      ( SRCBLK  := #AtributosDeUTs.Ruta,
        RET_VAL := #ReturnValor,
        DSTBLK  := "DB813_UTs_Ruta".UT[#VarTempUTs.NumeroUT].Ruta
      );

      L     201;  // 201 - Recibido Evento de nueva ruta para la UT
      T     "DB812_UTs_Control".UT[#VarTempUTs.NumeroUT].EstadoEventoRecibido;

//////////////////////////////////////////////////////////////////////
/// Inicio - Realizado 2017 07 06 // Control para Peticion de Ruta
      L     "DB812_UTs_Control".UT[#VarTempUTs.NumeroUT].MesaActual;
      L     #AtributosDeUTs.MesaDestino;
      <>I;
      JC    FinalGuardarRuta_EventoRecibido_CREA;

// Activar la Peticion de RUTA por llegada a su destino
      L     21;  // 21 - Generar Evento Pedir Ruta
      T     "DB812_UTs_Control".UT[#VarTempUTs.NumeroUT].EstadoGeneralUT;
      L     0;  // 0 - No Vale el Evento Recibido
      T     "DB812_UTs_Control".UT[#VarTempUTs.NumeroUT].EstadoEventoRecibido;

//////////////////////////////////////////////////////////////////////
// Final de Guardar Ruta
FinalGuardarRuta_EventoRecibido_CREA:NOP   0;



NETWORK
TITLE = ---- Final
/////////////////////////////////////////////////////////////////////////
/////////////////////////////////////////////////////////////////////////
/////////////////////////////////////////////////////////////////////////
// Se acabo el evento
Final_EventoRecibido_CREA:NOP   0;
      L     #P_Eventos;  // Recupero por donde voy en la lista de eventos
      LAR2;  // Regreso a buscar el siguiente evento
      JU    FinBucle_EventosRecibidos;



NETWORK
TITLE = Guardar Datos - Evento RUTA - Asignar ruta nueva a la UT
// Analisis del evento
//   - Inicializa variables de los atributos del Evento
//   - Buscar Atributos o Final del Evento
//   - Guardar datos del Evento
// Analisis de los atributos del Evento
//   - Mirar que atributo del Evento es
//   - Distribuir a recoger los datos del Evento
//   - Recoger el Atributo McKey
//   - Recoger el Atributo MesaActual
//   - Recoger el Atributo Nueva Ruta
GuardarDatos_EventoRecibido_RUTA:NOP   0;

/////////////////////////////////////////////////////////////////////////
/////////////////////////////////////////////////////////////////////////
/////////////////////////////////////////////////////////////////////////
// --- Guardar Datos del Evento Recibido


/////////////////////////////////////////////////////////////////////////
/////////////////////////////////////////////////////////////////////////
/////////////////////////////////////////////////////////////////////////
// --- Control de la Mesa Actual es Correcta
      L     #AtributosDeUTs.MesaActual;
      L     0;
      ==I;
      JC    FinControlMesa_EventoRecibido_RUTA;

      L     #AtributosDeUTs.MesaActual;  // Ver que mesa es
      L     "CTE_OffsetMesa";
      -I;
      T     #VarTempUTs.MesaActual;

      L     #VarTempUTs.MesaActual;  // Comprobar el numero de mesa
      L     1;  // No menor de 1
      <I;  // No es correcto
      JC    Final_EventoRecibido_RUTA;
      L     #VarTempUTs.MesaActual;
      L     "CTE_MaxMesas";  // No mayor que el parametro
      >I;  // No es correcto
      JC    Final_EventoRecibido_RUTA;

/////////////////////////////////////////////////////////////////////////
FinControlMesa_EventoRecibido_RUTA:NOP   0;


/////////////////////////////////////////////////////////////////////////
/////////////////////////////////////////////////////////////////////////
/////////////////////////////////////////////////////////////////////////
// --- Buscar UT en la Mesa Actual o por Mckey

      CALL  "FC720_BuscarUT_EnMesa"
      ( Mckey      := #AtributosDeUTs.Mckey,
        MesaActual := #VarTempUTs.MesaActual,
        NumeroUT   := #VarTempUTs.NumeroUT
      );

      L     #VarTempUTs.NumeroUT;
      L     0;
      ==I;  // No existe UT
      JC    Final_EventoRecibido_RUTA;



NETWORK
TITLE = ---- Accion del Evento
/////////////////////////////////////////////////////////////////////////
/////////////////////////////////////////////////////////////////////////
/////////////////////////////////////////////////////////////////////////
// Puntero a la UT, Marcar si es necesario -->
//           Actual = Destino = InterMedia --> Marcar la UT
// MODIFICACION --> 06/05/2013 (Alonso)

      SET;  // Reset - Recircular la Carga - Memoria del Retirar
      R     "DB812_UTs_Control".UT[#VarTempUTs.NumeroUT].AtributosDeLaUT.RecircularCarga;
      R     "DB812_UTs_Control".UT[#VarTempUTs.NumeroUT].AtributosDeLaUT.MemorizarRETI;

      L     "DB812_UTs_Control".UT[#VarTempUTs.NumeroUT].MesaActual;
      L     #AtributosDeUTs.MesaDestino;
      <>I;  // MesaActual <> MesaDestino ?
      JC    GuardarRutaRecibida_EventoRecibido_RUTA;

      L     #AtributosDeUTs.MesaDestino;
      L     #AtributosDeUTs.Ruta[0];
      ==I;
      JC    GuardarRutaRecibida_EventoRecibido_RUTA;

      SET;  // Set - Recircular la Carga
      S     "DB812_UTs_Control".UT[#VarTempUTs.NumeroUT].AtributosDeLaUT.RecircularCarga;


/////////////////////////////////////////////////////////////////////////
/////////////////////////////////////////////////////////////////////////
/////////////////////////////////////////////////////////////////////////
// --- Guardar ruta
GuardarRutaRecibida_EventoRecibido_RUTA:NOP   0;

      L     #AtributosDeUTs.MesaDestino;
      T     "DB812_UTs_Control".UT[#VarTempUTs.NumeroUT].MesaDestino;
      L     #AtributosDeUTs.MesaIntermedia;
      T     "DB812_UTs_Control".UT[#VarTempUTs.NumeroUT].MesaIntermedia;

      CALL  BLKMOV
      ( SRCBLK  := #AtributosDeUTs.Ruta,
        RET_VAL := #ReturnValor,
        DSTBLK  := "DB813_UTs_Ruta".UT[#VarTempUTs.NumeroUT].Ruta
      );

      L     201;  // 201 - Recibido Evento de Nueva Ruta para la UT
      T     "DB812_UTs_Control".UT[#VarTempUTs.NumeroUT].EstadoEventoRecibido;


/////////////////////////////////////////////////////////////////////////
/////////////////////////////////////////////////////////////////////////
//////////////////////////////////////////////////////////////////////
/// Inicio - Realizado 2017 07 06 // Control para Peticion de Ruta
      L     "DB812_UTs_Control".UT[#VarTempUTs.NumeroUT].MesaActual;
      L     #AtributosDeUTs.MesaDestino;
      <>I;
      JC    NoPedirRuta_EventoRecibido_RUTA;

      SET;  // Recircular la Carga ?
      A     "DB812_UTs_Control".UT[#VarTempUTs.NumeroUT].AtributosDeLaUT.RecircularCarga;
      JC    NoPedirRuta_EventoRecibido_RUTA;

// Activar la Peticion de RUTA por llegada a su destino
      L     21;  // 21 - Generar Evento Pedir Ruta
      T     "DB812_UTs_Control".UT[#VarTempUTs.NumeroUT].EstadoGeneralUT;
      L     0;  // 0 - No Vale el Evento Recibido
      T     "DB812_UTs_Control".UT[#VarTempUTs.NumeroUT].EstadoEventoRecibido;

//////////////////////////////////////////////////////////////////////
NoPedirRuta_EventoRecibido_RUTA:NOP   0;



NETWORK
TITLE = ---- Final
//////////////////////////////////////////////////////////////////////
//////////////////////////////////////////////////////////////////////
//////////////////////////////////////////////////////////////////////
// --- Se acabo el evento
Final_EventoRecibido_RUTA:NOP   0;
      L     #P_Eventos;  // Recupero por donde voy en la lista de eventos
      LAR2;  // Regreso a buscar el siguiente evento
      JU    FinBucle_EventosRecibidos;



NETWORK
TITLE = Guardar Datos - Evento DRUT - Asignar ruta nueva a la UT (Dinamica)
// Analisis del evento
//   - Inicializa variables de los atributos del Evento
//   - Buscar Atributos o Final del Evento
//   - Guardar datos del Evento
// Analisis de los atributos del Evento
//   - Mirar que atributo del Evento es
//   - Distribuir a recoger los datos del Evento
//   - Recoger el Atributo McKey
//   - Recoger el Atributo MesaActual
//   - Recoger el Atributo Nueva Ruta
GuardarDatos_EventoRecibido_DRUT:NOP   0;

/////////////////////////////////////////////////////////////////////////
/////////////////////////////////////////////////////////////////////////
/////////////////////////////////////////////////////////////////////////
// --- Guardar Datos del Evento Recibido


/////////////////////////////////////////////////////////////////////////
/////////////////////////////////////////////////////////////////////////
/////////////////////////////////////////////////////////////////////////
// --- Control de la Mesa Actual Recibida
      L     #AtributosDeUTs.MesaActual;
      L     0;
      ==I;
      JC    FinControlMesa_EventoRecibido_DRUT;

      L     #AtributosDeUTs.MesaActual;  // Ver que mesa es
      L     "CTE_OffsetMesa";
      -I;
      T     #VarTempUTs.MesaActual;

      L     #VarTempUTs.MesaActual;  // Comprobar el numero de mesa
      L     1;  // No menor de 1
      <I;  // No es correcto
      JC    Final_EventoRecibido_DRUT;
      L     #VarTempUTs.MesaActual;
      L     "CTE_MaxMesas";  // No mayor que el parametro
      >I;  // No es correcto
      JC    Final_EventoRecibido_DRUT;

/////////////////////////////////////////////////////////////////////////
FinControlMesa_EventoRecibido_DRUT:NOP   0;


/////////////////////////////////////////////////////////////////////////
/////////////////////////////////////////////////////////////////////////
/////////////////////////////////////////////////////////////////////////
// --- Buscar UT en la Mesa Actual o por Mckey

      CALL  "FC720_BuscarUT_EnMesa"
      ( Mckey      := #AtributosDeUTs.Mckey,
        MesaActual := #VarTempUTs.MesaActual,
        NumeroUT   := #VarTempUTs.NumeroUT
      );

      L     #VarTempUTs.NumeroUT;
      L     0;  // No existe UT
      ==I;
      JC    Final_EventoRecibido_DRUT;



NETWORK
TITLE = ---- Accion del Evento
/////////////////////////////////////////////////////////////////////////
/////////////////////////////////////////////////////////////////////////
/////////////////////////////////////////////////////////////////////////
// --- Guardar ruta

      L     #AtributosDeUTs.MesaDestino;
      T     "DB812_UTs_Control".UT[#VarTempUTs.NumeroUT].MesaDestino;
      L     #AtributosDeUTs.MesaIntermedia;
      T     "DB812_UTs_Control".UT[#VarTempUTs.NumeroUT].MesaIntermedia;

      CALL  BLKMOV
      ( SRCBLK  := #AtributosDeUTs.Ruta,
        RET_VAL := #ReturnValor,
        DSTBLK  := "DB813_UTs_Ruta".UT[#VarTempUTs.NumeroUT].Ruta
      );



NETWORK
TITLE = ---- Final
//////////////////////////////////////////////////////////////////////
//////////////////////////////////////////////////////////////////////
//////////////////////////////////////////////////////////////////////
// --- Se acabo el evento
Final_EventoRecibido_DRUT:NOP   0;
      L     #P_Eventos;  // Recupero por donde voy en la lista de eventos
      LAR2;  // Regreso a buscar el siguiente evento
      JU    FinBucle_EventosRecibidos;



NETWORK
TITLE = Guardar Datos - Evento RETI - Retirar la UT
// Analisis del evento
//   - Inicializa variables de los atributos del Evento
//   - Buscar Atributos o Final del Evento
//   - Guardar datos del Evento
// Analisis de los atributos del Evento
//   - Mirar que atributo del Evento es
//   - Distribuir a recoger los datos del Evento
//   - Recoger el Atributo McKey
//   - Recoger el Atributo MesaActual
GuardarDatos_EventoRecibido_RETI:NOP   0;

/////////////////////////////////////////////////////////////////////////
/////////////////////////////////////////////////////////////////////////
/////////////////////////////////////////////////////////////////////////
// --- Guardar Datos del Evento Recibido


/////////////////////////////////////////////////////////////////////////
/////////////////////////////////////////////////////////////////////////
/////////////////////////////////////////////////////////////////////////
// --- Control de Mesa Recibida
      L     #AtributosDeUTs.MesaActual;
      L     0;
      ==I;
      JC    FinControlMesa_EventoRecibido_RETI;

      L     #AtributosDeUTs.MesaActual;  // Ver que mesa es
      L     "CTE_OffsetMesa";
      -I;
      T     #VarTempUTs.MesaActual;

      L     #VarTempUTs.MesaActual;  // Comprobar el numero de mesa
      L     1;  // No menor de 1
      <I;  // No es correcto
      JC    Final_EventoRecibido_RETI;
      L     #VarTempUTs.MesaActual;
      L     "CTE_MaxMesas";  // No mayor que el parametro
      >I;  // No es correcto
      JC    Final_EventoRecibido_RETI;

/////////////////////////////////////////////////////////////////////////
FinControlMesa_EventoRecibido_RETI:NOP   0;


/////////////////////////////////////////////////////////////////////////
/////////////////////////////////////////////////////////////////////////
/////////////////////////////////////////////////////////////////////////
// --- Buscar UT en la Mesa Actual o Mckey
      CALL  "FC720_BuscarUT_EnMesa"
      ( Mckey      := #AtributosDeUTs.Mckey,
        MesaActual := #VarTempUTs.MesaActual,
        NumeroUT   := #VarTempUTs.NumeroUT
      );

      L     #VarTempUTs.NumeroUT;
      L     0;  // No existe UT
      ==I;
      JC    Final_EventoRecibido_RETI;



NETWORK
TITLE = ---- Accion del Evento
/////////////////////////////////////////////////////////////////////////
/////////////////////////////////////////////////////////////////////////
/////////////////////////////////////////////////////////////////////////
// --- Guardar datos
      L     #AtributosDeUTs.OrdenSalida;  // Sumar el numero de salida del Atributo
      L     210;  // 210 - Evento de Retirar la UT por S0
      +I;
      T     #VarTempUTs.SalidaEventoRETI;

      SET;  // Memorizar RETI - Ya memorizado
      A     "DB812_UTs_Control".UT[#VarTempUTs.NumeroUT].AtributosDeLaUT.MemorizarRETI;
      JC    ActivadaMemoria_EventoRecibido_RETI;

      L     #VarTempUTs.SalidaEventoRETI;  // EstadoEventoRecibido
      T     "DB812_UTs_Control".UT[#VarTempUTs.NumeroUT].EstadoEventoRecibido;

/////////////////////////////////////////////////////////////////////////
ActivadaMemoria_EventoRecibido_RETI:NOP   0;

      L     #VarTempUTs.SalidaEventoRETI;  // Mesa Intermeria --> Salida RETI
      T     "DB812_UTs_Control".UT[#VarTempUTs.NumeroUT].MesaIntermedia;

      SET;  // Set - Memorizar RETI
      S     "DB812_UTs_Control".UT[#VarTempUTs.NumeroUT].AtributosDeLaUT.MemorizarRETI;



